SPLINE
SPL {X  -146.770, Y  +318.818, Z    +0.000, E1  +325.496, E3 -247483.059}
SPL {X  -156.430, Y  +348.936, Z    +0.000, E1  +338.153, E3 -247499.791}
SPL {X  -159.088, Y  +365.539, Z    +0.000, E1  +347.196, E3 -247504.201}
SPL {X  -159.820, Y  +375.127, Z    +0.000, E1  +353.170, E3 -247505.625}
SPL {X  -159.990, Y  +382.134, Z    +0.000, E1  +357.935, E3 -247506.144}
SPL {X  -159.990, Y  +385.595, Z    +0.000, E1  +360.838, E3 -247506.258}
SPL {X  -159.990, Y  +390.176, Z    +0.000, E1  +366.367, E3 -247506.527}
SPL {X  -159.990, Y  +395.747, Z    +0.000, E1  +374.484, E3 -247507.153}
SPL {X  -159.990, Y  +402.387, Z    +0.000, E1  +384.140, E3 -247508.385}
SPL {X  -159.990, Y  +414.244, Z    +0.000, E1  +397.704, E3 -247512.018}
SPL {X  -159.990, Y  +460.468, Z    +0.000, E1  +416.751, E3 -247536.110}
SPL {X  -159.990, Y  +537.348, Z    +0.000, E1  +420.157, E3 -247606.121}
SPL {X  -159.990, Y  +545.972, Z    +0.000, E1  +420.143, E3 -247616.656}
SPL {X  -159.990, Y  +557.131, Z    +0.000, E1  +420.184, E3 -247630.170}
SPL {X  -159.990, Y  +569.073, Z    +0.000, E1  +420.153, E3 -247644.764}
SPL {X  -159.990, Y  +577.562, Z    +0.000, E1  +420.146, E3 -247655.104}
SPL {X  -159.990, Y  +585.415, Z    +0.000, E1  +420.147, E3 -247664.670}
SPL {X  -159.990, Y  +594.125, Z    +0.000, E1  +420.153, E3 -247675.256}
SPL {X  -159.990, Y  +602.716, Z    +0.000, E1  +420.150, E3 -247685.719}
SPL {X  -159.990, Y  +612.205, Z    +0.000, E1  +420.159, E3 -247697.255}
SPL {X  -159.990, Y  +624.752, Z    +0.000, E1  +420.194, E3 -247712.463}
SPL {X  -159.990, Y  +640.062, Z    +0.000, E1  +420.188, E3 -247731.127}
SPL {X  -159.990, Y  +652.098, Z    +0.000, E1  +420.153, E3 -247745.837}
SPL {X  -159.990, Y  +661.466, Z    +0.000, E1  +420.154, E3 -247757.248}
SPL {X  -159.963, Y  +674.441, Z    +0.000, E1  +420.189, E3 -247772.999}
SPL {X  -159.339, Y  +685.922, Z    +0.000, E1  +420.057, E3 -247787.677}
SPL {X  -158.381, Y  +694.132, Z    +0.000, E1  +419.909, E3 -247798.675}
SPL {X  -157.192, Y  +701.291, Z    +0.000, E1  +419.715, E3 -247808.645}
SPL {X  -155.426, Y  +709.440, Z    +0.000, E1  +419.459, E3 -247820.343}
SPL {X  -153.239, Y  +717.485, Z    +0.000, E1  +419.087, E3 -247832.388}
SPL {X  -150.608, Y  +725.483, Z    +0.000, E1  +418.677, E3 -247844.733}
SPL {X  -148.008, Y  +732.249, Z    +0.000, E1  +418.192, E3 -247855.600}
SPL {X  -145.943, Y  +737.055, Z    +0.000, E1  +417.829, E3 -247863.458}
SPL {X  -143.898, Y  +741.430, Z    +0.000, E1  +417.467, E3 -247870.728}
SPL {X  -140.579, Y  +747.882, Z    +0.000, E1  +416.895, E3 -247881.607}
SPL {X  -137.120, Y  +753.931, Z    +0.000, E1  +416.213, E3 -247892.067}
SPL {X  -120.054, Y  +777.254, Z    +0.000, E1  +409.463, E3 -247978.813}
ENDSPLINE

SPLINE
SPL {X  -141.034, Y  +747.040, Z    +0.000, E1  +398.619, E3 -248086.975}
SPL {X  -152.334, Y  +720.400, Z    +0.000, E1  +389.143, E3 -248106.429}
SPL {X  -157.190, Y  +701.303, Z    +0.000, E1  +380.164, E3 -248113.590}
SPL {X  -159.117, Y  +688.191, Z    +0.000, E1  +372.748, E3 -248116.622}
SPL {X  -159.875, Y  +677.561, Z    +0.000, E1  +366.083, E3 -248118.011}
SPL {X  -159.990, Y  +671.043, Z    +0.000, E1  +361.371, E3 -248118.415}
SPL {X  -159.990, Y  +669.269, Z    +0.000, E1  +359.855, E3 -248118.460}
SPL {X  -159.990, Y  +666.850, Z    +0.000, E1  +357.321, E3 -248118.543}
SPL {X  -159.990, Y  +662.495, Z    +0.000, E1  +351.318, E3 -248118.837}
SPL {X  -159.990, Y  +657.714, Z    +0.000, E1  +344.114, E3 -248119.398}
SPL {X  -159.990, Y  +651.822, Z    +0.000, E1  +335.261, E3 -248120.367}
SPL {X  -159.990, Y  +641.369, Z    +0.000, E1  +322.665, E3 -248123.205}
SPL {X  -159.990, Y  +598.251, Z    +0.000, E1  +304.104, E3 -248146.976}
SPL {X  -159.990, Y  +514.954, Z    +0.000, E1  +299.688, E3 -248220.772}
SPL {X  -159.990, Y  +505.641, Z    +0.000, E1  +299.707, E3 -248232.081}
SPL {X  -159.990, Y  +498.210, Z    +0.000, E1  +299.707, E3 -248241.074}
SPL {X  -159.990, Y  +488.988, Z    +0.000, E1  +299.693, E3 -248252.211}
SPL {X  -159.990, Y  +478.987, Z    +0.000, E1  +299.694, E3 -248264.314}
SPL {X  -159.990, Y  +468.796, Z    +0.000, E1  +299.698, E3 -248276.657}
SPL {X  -159.990, Y  +460.399, Z    +0.000, E1  +299.707, E3 -248286.834}
SPL {X  -159.990, Y  +453.289, Z    +0.000, E1  +299.707, E3 -248295.440}
SPL {X  -159.990, Y  +443.890, Z    +0.000, E1  +299.691, E3 -248306.793}
SPL {X  -159.990, Y  +437.910, Z    +0.000, E1  +300.175, E3 -248317.264}
ENDSPLINE

SPLINE
SPL {X  -159.990, Y  +447.165, Z    +0.000, E1  +303.287, E3 -248325.819}
ENDSPLINE

SPLINE
SPL {X  -159.990, Y  +436.354, Z    +0.000, E1  +302.683, E3 -248336.831}
SPL {X  -159.990, Y  +425.140, Z    +0.000, E1  +301.982, E3 -248347.266}
SPL {X  -159.990, Y  +412.625, Z    +0.000, E1  +301.150, E3 -248358.102}
SPL {X  -159.990, Y  +398.951, Z    +0.000, E1  +300.353, E3 -248369.973}
SPL {X  -159.990, Y  +389.564, Z    +0.000, E1  +300.093, E3 -248379.787}
SPL {X  -159.985, Y  +381.230, Z    +0.000, E1  +300.090, E3 -248390.054}
SPL {X  -159.702, Y  +372.900, Z    +0.000, E1  +300.135, E3 -248400.591}
SPL {X  -159.030, Y  +365.001, Z    +0.000, E1  +300.230, E3 -248410.994}
SPL {X  -158.029, Y  +357.528, Z    +0.000, E1  +300.403, E3 -248421.250}
SPL {X  -156.953, Y  +351.476, Z    +0.000, E1  +300.570, E3 -248429.803}
SPL {X  -155.503, Y  +344.875, Z    +0.000, E1  +300.798, E3 -248439.412}
SPL {X  -153.622, Y  +337.813, Z    +0.000, E1  +301.097, E3 -248450.006}
SPL {X  -151.786, Y  +331.925, Z    +0.000, E1  +301.419, E3 -248459.127}
SPL {X  -150.141, Y  +327.233, Z    +0.000, E1  +301.695, E3 -248466.535}
SPL {X  -148.134, Y  +322.059, Z    +0.000, E1  +302.038, E3 -248474.869}
SPL {X  -145.832, Y  +316.699, Z    +0.000, E1  +302.442, E3 -248483.703}
SPL {X  -143.160, Y  +311.071, Z    +0.000, E1  +302.918, E3 -248493.149}
SPL {X  -140.427, Y  +305.839, Z    +0.000, E1  +303.430, E3 -248502.110}
SPL {X  -137.611, Y  +300.891, Z    +0.000, E1  +303.950, E3 -248510.686}
SPL {X  -121.335, Y  +278.219, Z    +0.000, E1  +311.699, E3 -248609.032}
ENDSPLINE

SPLINE
SPL {X  -146.770, Y  +318.818, Z    +0.000, E1  +325.496, E3 -248708.866}
SPL {X  -156.430, Y  +348.936, Z    +0.000, E1  +338.153, E3 -248725.597}
SPL {X  -159.088, Y  +365.539, Z    +0.000, E1  +347.196, E3 -248730.008}
SPL {X  -159.921, Y  +377.798, Z    +0.000, E1  +354.872, E3 -248731.668}
SPL {X  -159.990, Y  +383.148, Z    +0.000, E1  +358.786, E3 -248731.996}
SPL {X  -159.990, Y  +384.761, Z    +0.000, E1  +360.138, E3 -248732.040}
SPL {X  -159.990, Y  +387.385, Z    +0.000, E1  +362.811, E3 -248732.142}
SPL {X  -159.990, Y  +391.439, Z    +0.000, E1  +368.259, E3 -248732.438}
SPL {X  -159.990, Y  +395.747, Z    +0.000, E1  +374.484, E3 -248732.959}
SPL {X  -159.990, Y  +402.387, Z    +0.000, E1  +384.140, E3 -248734.192}
SPL {X  -159.990, Y  +414.244, Z    +0.000, E1  +397.704, E3 -248737.825}
SPL {X  -159.990, Y  +460.468, Z    +0.000, E1  +416.751, E3 -248761.916}
SPL {X  -159.990, Y  +537.348, Z    +0.000, E1  +420.157, E3 -248831.928}
SPL {X  -159.990, Y  +549.907, Z    +0.000, E1  +420.183, E3 -248847.186}
SPL {X  -159.990, Y  +560.677, Z    +0.000, E1  +420.145, E3 -248860.357}
SPL {X  -159.990, Y  +569.073, Z    +0.000, E1  +420.153, E3 -248870.571}
SPL {X  -159.990, Y  +577.562, Z    +0.000, E1  +420.146, E3 -248880.911}
SPL {X  -159.990, Y  +585.415, Z    +0.000, E1  +420.147, E3 -248890.476}
SPL {X  -159.990, Y  +594.125, Z    +0.000, E1  +420.153, E3 -248901.063}
SPL {X  -159.990, Y  +602.716, Z    +0.000, E1  +420.150, E3 -248911.525}
SPL {X  -159.990, Y  +612.205, Z    +0.000, E1  +420.159, E3 -248923.062}
SPL {X  -159.990, Y  +620.604, Z    +0.000, E1  +420.153, E3 -248933.277}
SPL {X  -159.990, Y  +632.106, Z    +0.000, E1  +420.183, E3 -248947.254}
SPL {X  -159.990, Y  +643.341, Z    +0.000, E1  +420.148, E3 -248960.998}
SPL {X  -159.990, Y  +652.098, Z    +0.000, E1  +420.153, E3 -248971.643}
SPL {X  -159.990, Y  +661.466, Z    +0.000, E1  +420.154, E3 -248983.054}
SPL {X  -159.990, Y  +670.781, Z    +0.000, E1  +420.150, E3 -248994.402}
SPL {X  -159.839, Y  +678.445, Z    +0.000, E1  +420.123, E3 -249003.881}
SPL {X  -159.339, Y  +685.922, Z    +0.000, E1  +420.057, E3 -249013.484}
SPL {X  -158.381, Y  +694.132, Z    +0.000, E1  +419.909, E3 -249024.481}
SPL {X  -157.192, Y  +701.291, Z    +0.000, E1  +419.715, E3 -249034.451}
SPL {X  -155.426, Y  +709.440, Z    +0.000, E1  +419.459, E3 -249046.149}
SPL {X  -153.239, Y  +717.485, Z    +0.000, E1  +419.087, E3 -249058.194}
SPL {X  -151.467, Y  +723.022, Z    +0.000, E1  +418.780, E3 -249066.747}
SPL {X  -148.791, Y  +730.306, Z    +0.000, E1  +418.370, E3 -249078.212}
SPL {X  -145.943, Y  +737.055, Z    +0.000, E1  +417.829, E3 -249089.265}
SPL {X  -143.898, Y  +741.430, Z    +0.000, E1  +417.467, E3 -249096.534}
SPL {X  -141.624, Y  +745.927, Z    +0.000, E1  +417.045, E3 -249104.129}
SPL {X  -139.581, Y  +749.692, Z    +0.000, E1  +416.662, E3 -249110.576}
SPL {X  -137.120, Y  +753.931, Z    +0.000, E1  +416.213, E3 -249117.873}
SPL {X  -120.054, Y  +777.254, Z    +0.000, E1  +409.463, E3 -249204.619}
ENDSPLINE

SPLINE
SPL {X  -141.034, Y  +747.040, Z    +0.000, E1  +398.619, E3 -249312.781}
SPL {X  -152.334, Y  +720.400, Z    +0.000, E1  +389.143, E3 -249332.236}
SPL {X  -157.190, Y  +701.303, Z    +0.000, E1  +380.164, E3 -249339.396}
SPL {X  -159.117, Y  +688.191, Z    +0.000, E1  +372.748, E3 -249342.428}
SPL {X  -159.875, Y  +677.561, Z    +0.000, E1  +366.083, E3 -249343.818}
SPL {X  -159.990, Y  +669.975, Z    +0.000, E1  +360.595, E3 -249344.249}
SPL {X  -159.990, Y  +666.850, Z    +0.000, E1  +357.321, E3 -249344.349}
SPL {X  -159.990, Y  +662.495, Z    +0.000, E1  +351.318, E3 -249344.644}
SPL {X  -159.990, Y  +657.714, Z    +0.000, E1  +344.114, E3 -249345.205}
SPL {X  -159.990, Y  +651.822, Z    +0.000, E1  +335.261, E3 -249346.173}
SPL {X  -159.990, Y  +641.369, Z    +0.000, E1  +322.665, E3 -249349.011}
SPL {X  -159.990, Y  +598.251, Z    +0.000, E1  +304.104, E3 -249372.782}
SPL {X  -159.990, Y  +514.954, Z    +0.000, E1  +299.688, E3 -249446.578}
SPL {X  -159.990, Y  +505.641, Z    +0.000, E1  +299.707, E3 -249457.887}
SPL {X  -159.990, Y  +498.210, Z    +0.000, E1  +299.707, E3 -249466.881}
SPL {X  -159.990, Y  +488.988, Z    +0.000, E1  +299.693, E3 -249478.017}
SPL {X  -159.990, Y  +478.987, Z    +0.000, E1  +299.694, E3 -249490.120}
SPL {X  -159.990, Y  +468.796, Z    +0.000, E1  +299.698, E3 -249502.464}
SPL {X  -159.990, Y  +460.399, Z    +0.000, E1  +299.707, E3 -249512.641}
SPL {X  -159.990, Y  +453.289, Z    +0.000, E1  +299.707, E3 -249521.246}
SPL {X  -159.990, Y  +443.890, Z    +0.000, E1  +299.691, E3 -249532.600}
SPL {X  -159.990, Y  +437.910, Z    +0.000, E1  +300.175, E3 -249543.070}
ENDSPLINE

SPLINE
SPL {X  -159.990, Y  +447.165, Z    +0.000, E1  +303.287, E3 -249551.626}
ENDSPLINE

SPLINE
SPL {X  -159.990, Y  +436.354, Z    +0.000, E1  +302.683, E3 -249562.637}
SPL {X  -159.990, Y  +425.140, Z    +0.000, E1  +301.982, E3 -249573.072}
SPL {X  -159.990, Y  +412.625, Z    +0.000, E1  +301.150, E3 -249583.908}
SPL {X  -159.990, Y  +398.951, Z    +0.000, E1  +300.353, E3 -249595.780}
SPL {X  -159.990, Y  +389.564, Z    +0.000, E1  +300.093, E3 -249605.594}
SPL {X  -159.985, Y  +381.230, Z    +0.000, E1  +300.090, E3 -249615.861}
SPL {X  -159.702, Y  +372.900, Z    +0.000, E1  +300.135, E3 -249626.398}
SPL {X  -159.030, Y  +365.001, Z    +0.000, E1  +300.230, E3 -249636.801}
SPL {X  -157.449, Y  +354.098, Z    +0.000, E1  +300.447, E3 -249651.800}
SPL {X  -155.503, Y  +344.875, Z    +0.000, E1  +300.798, E3 -249665.219}
SPL {X  -153.622, Y  +337.813, Z    +0.000, E1  +301.097, E3 -249675.812}
SPL {X  -150.877, Y  +329.275, Z    +0.000, E1  +301.527, E3 -249689.037}
SPL {X  -148.134, Y  +322.059, Z    +0.000, E1  +302.038, E3 -249700.675}
SPL {X  -145.832, Y  +316.699, Z    +0.000, E1  +302.442, E3 -249709.510}
SPL {X  -143.160, Y  +311.071, Z    +0.000, E1  +302.918, E3 -249718.955}
SPL {X  -140.427, Y  +305.839, Z    +0.000, E1  +303.430, E3 -249727.916}
SPL {X  -137.611, Y  +300.891, Z    +0.000, E1  +303.950, E3 -249736.492}
SPL {X  -121.335, Y  +278.219, Z    +0.000, E1  +311.699, E3 -249834.838}
ENDSPLINE

SPLINE
SPL {X  -146.770, Y  +318.818, Z    +0.000, E1  +325.496, E3 -249934.672}
SPL {X  -156.430, Y  +348.936, Z    +0.000, E1  +338.153, E3 -249951.404}
SPL {X  -159.088, Y  +365.539, Z    +0.000, E1  +347.196, E3 -249955.814}
SPL {X  -159.820, Y  +375.127, Z    +0.000, E1  +353.170, E3 -249957.238}
SPL {X  -159.990, Y  +382.134, Z    +0.000, E1  +357.935, E3 -249957.757}
SPL {X  -159.990, Y  +385.595, Z    +0.000, E1  +360.838, E3 -249957.871}
SPL {X  -159.990, Y  +390.176, Z    +0.000, E1  +366.367, E3 -249958.140}
SPL {X  -159.990, Y  +395.747, Z    +0.000, E1  +374.484, E3 -249958.766}
SPL {X  -159.990, Y  +404.190, Z    +0.000, E1  +386.444, E3 -249960.448}
SPL {X  -159.990, Y  +418.143, Z    +0.000, E1  +401.167, E3 -249965.041}
SPL {X  -159.990, Y  +460.468, Z    +0.000, E1  +416.751, E3 -249987.723}
SPL {X  -159.990, Y  +537.348, Z    +0.000, E1  +420.157, E3 -250057.734}
SPL {X  -159.990, Y  +549.907, Z    +0.000, E1  +420.183, E3 -250072.992}
SPL {X  -159.990, Y  +560.677, Z    +0.000, E1  +420.145, E3 -250086.163}
SPL {X  -159.990, Y  +569.073, Z    +0.000, E1  +420.153, E3 -250096.377}
SPL {X  -159.990, Y  +581.828, Z    +0.000, E1  +420.191, E3 -250111.837}
SPL {X  -159.990, Y  +594.125, Z    +0.000, E1  +420.153, E3 -250126.869}
SPL {X  -159.990, Y  +602.716, Z    +0.000, E1  +420.150, E3 -250137.332}
SPL {X  -159.990, Y  +612.205, Z    +0.000, E1  +420.159, E3 -250148.868}
SPL {X  -159.990, Y  +620.604, Z    +0.000, E1  +420.153, E3 -250159.084}
SPL {X  -159.990, Y  +632.106, Z    +0.000, E1  +420.183, E3 -250173.061}
SPL {X  -159.990, Y  +643.341, Z    +0.000, E1  +420.148, E3 -250186.804}
SPL {X  -159.990, Y  +652.098, Z    +0.000, E1  +420.153, E3 -250197.449}
SPL {X  -159.990, Y  +661.466, Z    +0.000, E1  +420.154, E3 -250208.861}
SPL {X  -159.990, Y  +670.781, Z    +0.000, E1  +420.150, E3 -250220.209}
SPL {X  -159.839, Y  +678.445, Z    +0.000, E1  +420.123, E3 -250229.688}
SPL {X  -159.339, Y  +685.922, Z    +0.000, E1  +420.057, E3 -250239.290}
SPL {X  -158.381, Y  +694.132, Z    +0.000, E1  +419.909, E3 -250250.287}
SPL {X  -157.192, Y  +701.291, Z    +0.000, E1  +419.715, E3 -250260.258}
SPL {X  -155.426, Y  +709.440, Z    +0.000, E1  +419.459, E3 -250271.956}
SPL {X  -153.239, Y  +717.485, Z    +0.000, E1  +419.087, E3 -250284.001}
SPL {X  -150.608, Y  +725.483, Z    +0.000, E1  +418.677, E3 -250296.346}
SPL {X  -148.008, Y  +732.249, Z    +0.000, E1  +418.192, E3 -250307.213}
SPL {X  -145.943, Y  +737.055, Z    +0.000, E1  +417.829, E3 -250315.071}
SPL {X  -143.898, Y  +741.430, Z    +0.000, E1  +417.467, E3 -250322.341}
SPL {X  -141.624, Y  +745.927, Z    +0.000, E1  +417.045, E3 -250329.936}
SPL {X  -139.581, Y  +749.692, Z    +0.000, E1  +416.662, E3 -250336.383}
SPL {X  -137.120, Y  +753.931, Z    +0.000, E1  +416.213, E3 -250343.680}
SPL {X  -120.054, Y  +777.254, Z    +0.000, E1  +409.463, E3 -250430.426}
ENDSPLINE

SPLINE
SPL {X  -141.034, Y  +747.040, Z    +0.000, E1  +398.619, E3 -250538.588}
SPL {X  -152.334, Y  +720.400, Z    +0.000, E1  +389.143, E3 -250558.042}
SPL {X  -157.190, Y  +701.303, Z    +0.000, E1  +380.164, E3 -250565.203}
SPL {X  -159.460, Y  +684.516, Z    +0.000, E1  +370.556, E3 -250568.798}
SPL {X  -159.938, Y  +675.597, Z    +0.000, E1  +364.669, E3 -250569.805}
SPL {X  -159.990, Y  +671.043, Z    +0.000, E1  +361.371, E3 -250570.028}
SPL {X  -159.990, Y  +669.269, Z    +0.000, E1  +359.855, E3 -250570.073}
SPL {X  -159.990, Y  +666.850, Z    +0.000, E1  +357.321, E3 -250570.156}
SPL {X  -159.990, Y  +662.495, Z    +0.000, E1  +351.318, E3 -250570.450}
SPL {X  -159.990, Y  +657.714, Z    +0.000, E1  +344.114, E3 -250571.011}
SPL {X  -159.990, Y  +651.822, Z    +0.000, E1  +335.261, E3 -250571.979}
SPL {X  -159.990, Y  +641.369, Z    +0.000, E1  +322.665, E3 -250574.818}
SPL {X  -159.990, Y  +598.251, Z    +0.000, E1  +304.104, E3 -250598.589}
SPL {X  -159.990, Y  +514.954, Z    +0.000, E1  +299.688, E3 -250672.384}
SPL {X  -159.990, Y  +505.641, Z    +0.000, E1  +299.707, E3 -250683.694}
SPL {X  -159.990, Y  +498.210, Z    +0.000, E1  +299.707, E3 -250692.687}
SPL {X  -159.990, Y  +488.988, Z    +0.000, E1  +299.693, E3 -250703.824}
SPL {X  -159.990, Y  +478.987, Z    +0.000, E1  +299.694, E3 -250715.926}
SPL {X  -159.990, Y  +468.796, Z    +0.000, E1  +299.698, E3 -250728.270}
SPL {X  -159.990, Y  +456.606, Z    +0.000, E1  +299.670, E3 -250742.976}
SPL {X  -159.990, Y  +443.890, Z    +0.000, E1  +299.691, E3 -250758.406}
SPL {X  -159.990, Y  +437.910, Z    +0.000, E1  +300.175, E3 -250768.877}
ENDSPLINE

SPLINE
SPL {X  -159.990, Y  +447.165, Z    +0.000, E1  +303.287, E3 -250777.432}
ENDSPLINE

SPLINE
SPL {X  -159.990, Y  +436.354, Z    +0.000, E1  +302.683, E3 -250788.443}
SPL {X  -159.990, Y  +425.140, Z    +0.000, E1  +301.982, E3 -250798.879}
SPL {X  -159.990, Y  +412.625, Z    +0.000, E1  +301.150, E3 -250809.715}
SPL {X  -159.990, Y  +398.951, Z    +0.000, E1  +300.353, E3 -250821.586}
SPL {X  -159.990, Y  +389.564, Z    +0.000, E1  +300.093, E3 -250831.400}
SPL {X  -159.985, Y  +381.230, Z    +0.000, E1  +300.090, E3 -250841.667}
SPL {X  -159.702, Y  +372.900, Z    +0.000, E1  +300.135, E3 -250852.204}
SPL {X  -159.030, Y  +365.001, Z    +0.000, E1  +300.230, E3 -250862.607}
SPL {X  -158.029, Y  +357.528, Z    +0.000, E1  +300.403, E3 -250872.862}
SPL {X  -156.953, Y  +351.476, Z    +0.000, E1  +300.570, E3 -250881.416}
SPL {X  -155.503, Y  +344.875, Z    +0.000, E1  +300.798, E3 -250891.025}
SPL {X  -153.622, Y  +337.813, Z    +0.000, E1  +301.097, E3 -250901.619}
SPL {X  -150.877, Y  +329.275, Z    +0.000, E1  +301.527, E3 -250914.843}
SPL {X  -148.134, Y  +322.059, Z    +0.000, E1  +302.038, E3 -250926.482}
SPL {X  -145.832, Y  +316.699, Z    +0.000, E1  +302.442, E3 -250935.316}
SPL {X  -143.160, Y  +311.071, Z    +0.000, E1  +302.918, E3 -250944.762}
SPL {X  -140.427, Y  +305.839, Z    +0.000, E1  +303.430, E3 -250953.723}
SPL {X  -137.611, Y  +300.891, Z    +0.000, E1  +303.950, E3 -250962.299}
SPL {X  -121.335, Y  +278.219, Z    +0.000, E1  +311.699, E3 -251060.645}
ENDSPLINE

SPLINE
SPL {X  -146.770, Y  +318.818, Z    +0.000, E1  +325.496, E3 -251160.479}
SPL {X  -156.430, Y  +348.936, Z    +0.000, E1  +338.153, E3 -251177.210}
SPL {X  -159.088, Y  +365.539, Z    +0.000, E1  +347.196, E3 -251181.621}
SPL {X  -159.921, Y  +377.798, Z    +0.000, E1  +354.872, E3 -251183.281}
SPL {X  -159.990, Y  +384.169, Z    +0.000, E1  +359.534, E3 -251183.637}
SPL {X  -159.990, Y  +386.366, Z    +0.000, E1  +361.774, E3 -251183.701}
SPL {X  -159.990, Y  +390.176, Z    +0.000, E1  +366.367, E3 -251183.947}
SPL {X  -159.990, Y  +395.747, Z    +0.000, E1  +374.484, E3 -251184.572}
SPL {X  -159.990, Y  +402.387, Z    +0.000, E1  +384.140, E3 -251185.805}
SPL {X  -159.990, Y  +414.244, Z    +0.000, E1  +397.704, E3 -251189.438}
SPL {X  -159.990, Y  +460.468, Z    +0.000, E1  +416.751, E3 -251213.529}
SPL {X  -159.990, Y  +537.348, Z    +0.000, E1  +420.157, E3 -251283.541}
SPL {X  -159.990, Y  +545.972, Z    +0.000, E1  +420.143, E3 -251294.075}
SPL {X  -159.990, Y  +557.131, Z    +0.000, E1  +420.184, E3 -251307.589}
SPL {X  -159.990, Y  +569.073, Z    +0.000, E1  +420.153, E3 -251322.184}
SPL {X  -159.990, Y  +581.828, Z    +0.000, E1  +420.191, E3 -251337.643}
SPL {X  -159.990, Y  +594.125, Z    +0.000, E1  +420.153, E3 -251352.676}
SPL {X  -159.990, Y  +602.716, Z    +0.000, E1  +420.150, E3 -251363.138}
SPL {X  -159.990, Y  +612.205, Z    +0.000, E1  +420.159, E3 -251374.675}
SPL {X  -159.990, Y  +624.752, Z    +0.000, E1  +420.194, E3 -251389.883}
SPL {X  -159.990, Y  +640.062, Z    +0.000, E1  +420.188, E3 -251408.546}
SPL {X  -159.990, Y  +652.098, Z    +0.000, E1  +420.153, E3 -251423.256}
SPL {X  -159.990, Y  +661.466, Z    +0.000, E1  +420.154, E3 -251434.667}
SPL {X  -159.963, Y  +674.441, Z    +0.000, E1  +420.189, E3 -251450.418}
SPL {X  -159.339, Y  +685.922, Z    +0.000, E1  +420.057, E3 -251465.097}
SPL {X  -158.381, Y  +694.132, Z    +0.000, E1  +419.909, E3 -251476.094}
SPL {X  -156.712, Y  +703.719, Z    +0.000, E1  +419.674, E3 -251489.459}
SPL {X  -154.922, Y  +711.450, Z    +0.000, E1  +419.348, E3 -251500.775}
SPL {X  -153.239, Y  +717.485, Z    +0.000, E1  +419.087, E3 -251509.807}
SPL {X  -150.608, Y  +725.483, Z    +0.000, E1  +418.677, E3 -251522.153}
SPL {X  -148.008, Y  +732.249, Z    +0.000, E1  +418.192, E3 -251533.019}
SPL {X  -145.943, Y  +737.055, Z    +0.000, E1  +417.829, E3 -251540.878}
SPL {X  -143.898, Y  +741.430, Z    +0.000, E1  +417.467, E3 -251548.147}
SPL {X  -141.624, Y  +745.927, Z    +0.000, E1  +417.045, E3 -251555.742}
SPL {X  -139.581, Y  +749.692, Z    +0.000, E1  +416.662, E3 -251562.189}
SPL {X  -137.120, Y  +753.931, Z    +0.000, E1  +416.213, E3 -251569.486}
SPL {X  -120.054, Y  +777.254, Z    +0.000, E1  +409.463, E3 -251656.232}
ENDSPLINE

SPLINE
SPL {X  -141.034, Y  +747.040, Z    +0.000, E1  +398.619, E3 -251764.394}
SPL {X  -152.334, Y  +720.400, Z    +0.000, E1  +389.143, E3 -251783.848}
SPL {X  -157.190, Y  +701.303, Z    +0.000, E1  +380.164, E3 -251791.009}
SPL {X  -159.117, Y  +688.191, Z    +0.000, E1  +372.748, E3 -251794.041}
SPL {X  -159.875, Y  +677.561, Z    +0.000, E1  +366.083, E3 -251795.431}
SPL {X  -159.990, Y  +669.975, Z    +0.000, E1  +360.595, E3 -251795.862}
SPL {X  -159.990, Y  +666.850, Z    +0.000, E1  +357.321, E3 -251795.962}
SPL {X  -159.990, Y  +662.495, Z    +0.000, E1  +351.318, E3 -251796.257}
SPL {X  -159.990, Y  +657.714, Z    +0.000, E1  +344.114, E3 -251796.818}
SPL {X  -159.990, Y  +651.822, Z    +0.000, E1  +335.261, E3 -251797.786}
SPL {X  -159.990, Y  +641.369, Z    +0.000, E1  +322.665, E3 -251800.624}
SPL {X  -159.990, Y  +598.251, Z    +0.000, E1  +304.104, E3 -251824.395}
SPL {X  -159.990, Y  +514.954, Z    +0.000, E1  +299.688, E3 -251898.191}
SPL {X  -159.990, Y  +505.641, Z    +0.000, E1  +299.707, E3 -251909.500}
SPL {X  -159.990, Y  +498.210, Z    +0.000, E1  +299.707, E3 -251918.494}
SPL {X  -159.990, Y  +488.988, Z    +0.000, E1  +299.693, E3 -251929.630}
SPL {X  -159.990, Y  +478.987, Z    +0.000, E1  +299.694, E3 -251941.733}
SPL {X  -159.990, Y  +468.796, Z    +0.000, E1  +299.698, E3 -251954.077}
SPL {X  -159.990, Y  +456.606, Z    +0.000, E1  +299.670, E3 -251968.782}
SPL {X  -159.990, Y  +443.890, Z    +0.000, E1  +299.691, E3 -251984.212}
SPL {X  -159.990, Y  +437.910, Z    +0.000, E1  +300.175, E3 -251994.683}
ENDSPLINE

SPLINE
SPL {X  -159.990, Y  +447.165, Z    +0.000, E1  +303.287, E3 -252003.238}
ENDSPLINE

SPLINE
SPL {X  -159.990, Y  +436.354, Z    +0.000, E1  +302.683, E3 -252014.250}
SPL {X  -159.990, Y  +425.140, Z    +0.000, E1  +301.982, E3 -252024.685}
SPL {X  -159.990, Y  +412.625, Z    +0.000, E1  +301.150, E3 -252035.521}
SPL {X  -159.990, Y  +398.951, Z    +0.000, E1  +300.353, E3 -252047.393}
SPL {X  -159.990, Y  +389.564, Z    +0.000, E1  +300.093, E3 -252057.207}
SPL {X  -159.985, Y  +381.230, Z    +0.000, E1  +300.090, E3 -252067.474}
SPL {X  -159.702, Y  +372.900, Z    +0.000, E1  +300.135, E3 -252078.011}
SPL {X  -159.030, Y  +365.001, Z    +0.000, E1  +300.230, E3 -252088.413}
SPL {X  -158.029, Y  +357.528, Z    +0.000, E1  +300.403, E3 -252098.669}
SPL {X  -156.953, Y  +351.476, Z    +0.000, E1  +300.570, E3 -252107.222}
SPL {X  -155.503, Y  +344.875, Z    +0.000, E1  +300.798, E3 -252116.832}
SPL {X  -153.622, Y  +337.813, Z    +0.000, E1  +301.097, E3 -252127.425}
SPL {X  -151.786, Y  +331.925, Z    +0.000, E1  +301.419, E3 -252136.546}
SPL {X  -150.141, Y  +327.233, Z    +0.000, E1  +301.695, E3 -252143.955}
SPL {X  -148.134, Y  +322.059, Z    +0.000, E1  +302.038, E3 -252152.288}
SPL {X  -145.832, Y  +316.699, Z    +0.000, E1  +302.442, E3 -252161.123}
SPL {X  -143.160, Y  +311.071, Z    +0.000, E1  +302.918, E3 -252170.568}
SPL {X  -140.427, Y  +305.839, Z    +0.000, E1  +303.430, E3 -252179.529}
SPL {X  -137.611, Y  +300.891, Z    +0.000, E1  +303.950, E3 -252188.105}
SPL {X  -121.335, Y  +278.219, Z    +0.000, E1  +311.699, E3 -252286.451}
ENDSPLINE

SPLINE
SPL {X  -146.770, Y  +318.818, Z    +0.000, E1  +325.496, E3 -252386.285}
SPL {X  -156.430, Y  +348.936, Z    +0.000, E1  +338.153, E3 -252403.016}
SPL {X  -159.088, Y  +365.539, Z    +0.000, E1  +347.196, E3 -252407.427}
SPL {X  -159.921, Y  +377.798, Z    +0.000, E1  +354.872, E3 -252409.087}
SPL {X  -159.990, Y  +384.169, Z    +0.000, E1  +359.534, E3 -252409.443}
SPL {X  -159.990, Y  +386.366, Z    +0.000, E1  +361.774, E3 -252409.507}
SPL {X  -159.990, Y  +390.176, Z    +0.000, E1  +366.367, E3 -252409.753}
SPL {X  -159.990, Y  +395.747, Z    +0.000, E1  +374.484, E3 -252410.379}
SPL {X  -159.990, Y  +402.387, Z    +0.000, E1  +384.140, E3 -252411.611}
SPL {X  -159.990, Y  +414.244, Z    +0.000, E1  +397.704, E3 -252415.244}
SPL {X  -159.990, Y  +460.468, Z    +0.000, E1  +416.751, E3 -252439.336}
SPL {X  -159.990, Y  +537.348, Z    +0.000, E1  +420.157, E3 -252509.347}
SPL {X  -159.990, Y  +545.972, Z    +0.000, E1  +420.143, E3 -252519.881}
SPL {X  -159.990, Y  +557.131, Z    +0.000, E1  +420.184, E3 -252533.396}
SPL {X  -159.990, Y  +569.073, Z    +0.000, E1  +420.153, E3 -252547.990}
SPL {X  -159.990, Y  +577.562, Z    +0.000, E1  +420.146, E3 -252558.330}
SPL {X  -159.990, Y  +585.415, Z    +0.000, E1  +420.147, E3 -252567.896}
SPL {X  -159.990, Y  +594.125, Z    +0.000, E1  +420.153, E3 -252578.482}
SPL {X  -159.990, Y  +602.716, Z    +0.000, E1  +420.150, E3 -252588.945}
SPL {X  -159.990, Y  +612.205, Z    +0.000, E1  +420.159, E3 -252600.481}
SPL {X  -159.990, Y  +624.752, Z    +0.000, E1  +420.194, E3 -252615.689}
SPL {X  -159.990, Y  +640.062, Z    +0.000, E1  +420.188, E3 -252634.353}
SPL {X  -159.990, Y  +652.098, Z    +0.000, E1  +420.153, E3 -252649.062}
SPL {X  -159.990, Y  +661.466, Z    +0.000, E1  +420.154, E3 -252660.474}
SPL {X  -159.990, Y  +670.781, Z    +0.000, E1  +420.150, E3 -252671.821}
SPL {X  -159.839, Y  +678.445, Z    +0.000, E1  +420.123, E3 -252681.301}
SPL {X  -159.339, Y  +685.922, Z    +0.000, E1  +420.057, E3 -252690.903}
SPL {X  -158.381, Y  +694.132, Z    +0.000, E1  +419.909, E3 -252701.900}
SPL {X  -156.712, Y  +703.719, Z    +0.000, E1  +419.674, E3 -252715.265}
SPL {X  -154.922, Y  +711.450, Z    +0.000, E1  +419.348, E3 -252726.581}
SPL {X  -153.239, Y  +717.485, Z    +0.000, E1  +419.087, E3 -252735.614}
SPL {X  -150.608, Y  +725.483, Z    +0.000, E1  +418.677, E3 -252747.959}
SPL {X  -148.008, Y  +732.249, Z    +0.000, E1  +418.192, E3 -252758.826}
SPL {X  -145.943, Y  +737.055, Z    +0.000, E1  +417.829, E3 -252766.684}
SPL {X  -143.898, Y  +741.430, Z    +0.000, E1  +417.467, E3 -252773.954}
SPL {X  -141.624, Y  +745.927, Z    +0.000, E1  +417.045, E3 -252781.549}
SPL {X  -139.581, Y  +749.692, Z    +0.000, E1  +416.662, E3 -252787.995}
SPL {X  -137.120, Y  +753.931, Z    +0.000, E1  +416.213, E3 -252795.293}
SPL {X  -120.054, Y  +777.254, Z    +0.000, E1  +409.463, E3 -252882.039}
ENDSPLINE

SPLINE
SPL {X  -141.034, Y  +747.040, Z    +0.000, E1  +398.619, E3 -252990.201}
SPL {X  -152.334, Y  +720.400, Z    +0.000, E1  +389.143, E3 -253009.655}
SPL {X  -157.190, Y  +701.303, Z    +0.000, E1  +380.164, E3 -253016.816}
SPL {X  -159.117, Y  +688.191, Z    +0.000, E1  +372.748, E3 -253019.848}
SPL {X  -159.875, Y  +677.561, Z    +0.000, E1  +366.083, E3 -253021.237}
SPL {X  -159.990, Y  +671.043, Z    +0.000, E1  +361.371, E3 -253021.641}
SPL {X  -159.990, Y  +668.657, Z    +0.000, E1  +359.332, E3 -253021.702}
SPL {X  -159.990, Y  +665.812, Z    +0.000, E1  +355.875, E3 -253021.813}
SPL {X  -159.990, Y  +662.495, Z    +0.000, E1  +351.318, E3 -253022.063}
SPL {X  -159.990, Y  +657.714, Z    +0.000, E1  +344.114, E3 -253022.624}
SPL {X  -159.990, Y  +651.822, Z    +0.000, E1  +335.261, E3 -253023.592}
SPL {X  -159.990, Y  +641.369, Z    +0.000, E1  +322.665, E3 -253026.431}
SPL {X  -159.990, Y  +598.251, Z    +0.000, E1  +304.104, E3 -253050.202}
SPL {X  -159.990, Y  +514.954, Z    +0.000, E1  +299.688, E3 -253123.997}
SPL {X  -159.990, Y  +505.641, Z    +0.000, E1  +299.707, E3 -253135.306}
SPL {X  -159.990, Y  +498.210, Z    +0.000, E1  +299.707, E3 -253144.300}
SPL {X  -159.990, Y  +488.988, Z    +0.000, E1  +299.693, E3 -253155.437}
SPL {X  -159.990, Y  +478.987, Z    +0.000, E1  +299.694, E3 -253167.539}
SPL {X  -159.990, Y  +468.796, Z    +0.000, E1  +299.698, E3 -253179.883}
SPL {X  -159.990, Y  +456.606, Z    +0.000, E1  +299.670, E3 -253194.589}
SPL {X  -159.990, Y  +443.890, Z    +0.000, E1  +299.691, E3 -253210.019}
SPL {X  -159.990, Y  +437.910, Z    +0.000, E1  +300.175, E3 -253220.490}
ENDSPLINE

SPLINE
SPL {X  -159.990, Y  +447.165, Z    +0.000, E1  +303.287, E3 -253229.045}
ENDSPLINE

SPLINE
SPL {X  -159.990, Y  +436.354, Z    +0.000, E1  +302.683, E3 -253240.056}
SPL {X  -159.990, Y  +425.140, Z    +0.000, E1  +301.982, E3 -253250.492}
SPL {X  -159.990, Y  +412.625, Z    +0.000, E1  +301.150, E3 -253261.328}
SPL {X  -159.990, Y  +398.951, Z    +0.000, E1  +300.353, E3 -253273.199}
SPL {X  -159.990, Y  +389.564, Z    +0.000, E1  +300.093, E3 -253283.013}
SPL {X  -159.985, Y  +381.230, Z    +0.000, E1  +300.090, E3 -253293.280}
SPL {X  -159.702, Y  +372.900, Z    +0.000, E1  +300.135, E3 -253303.817}
SPL {X  -159.030, Y  +365.001, Z    +0.000, E1  +300.230, E3 -253314.220}
SPL {X  -157.449, Y  +354.098, Z    +0.000, E1  +300.447, E3 -253329.220}
SPL {X  -155.503, Y  +344.875, Z    +0.000, E1  +300.798, E3 -253342.638}
SPL {X  -153.622, Y  +337.813, Z    +0.000, E1  +301.097, E3 -253353.231}
SPL {X  -150.877, Y  +329.275, Z    +0.000, E1  +301.527, E3 -253366.456}
SPL {X  -148.134, Y  +322.059, Z    +0.000, E1  +302.038, E3 -253378.095}
SPL {X  -145.832, Y  +316.699, Z    +0.000, E1  +302.442, E3 -253386.929}
SPL {X  -143.160, Y  +311.071, Z    +0.000, E1  +302.918, E3 -253396.374}
SPL {X  -140.427, Y  +305.839, Z    +0.000, E1  +303.430, E3 -253405.336}
SPL {X  -137.611, Y  +300.891, Z    +0.000, E1  +303.950, E3 -253413.912}
SPL {X  -121.335, Y  +278.219, Z    +0.000, E1  +311.699, E3 -253512.258}
ENDSPLINE

SPLINE
SPL {X  -146.770, Y  +318.818, Z    +0.000, E1  +325.496, E3 -253612.092}
SPL {X  -156.430, Y  +348.936, Z    +0.000, E1  +338.153, E3 -253628.823}
SPL {X  -159.088, Y  +365.539, Z    +0.000, E1  +347.196, E3 -253633.234}
SPL {X  -159.820, Y  +375.127, Z    +0.000, E1  +353.170, E3 -253634.657}
SPL {X  -159.990, Y  +382.134, Z    +0.000, E1  +357.935, E3 -253635.176}
SPL {X  -159.990, Y  +385.595, Z    +0.000, E1  +360.838, E3 -253635.291}
SPL {X  -159.990, Y  +390.176, Z    +0.000, E1  +366.367, E3 -253635.560}
SPL {X  -159.990, Y  +395.747, Z    +0.000, E1  +374.484, E3 -253636.185}
SPL {X  -159.990, Y  +402.387, Z    +0.000, E1  +384.140, E3 -253637.418}
SPL {X  -159.990, Y  +413.408, Z    +0.000, E1  +396.965, E3 -253640.719}
SPL {X  -159.990, Y  +455.723, Z    +0.000, E1  +415.803, E3 -253662.561}
SPL {X  -159.990, Y  +537.348, Z    +0.000, E1  +420.157, E3 -253735.154}
SPL {X  -159.990, Y  +545.972, Z    +0.000, E1  +420.143, E3 -253745.688}
SPL {X  -159.990, Y  +557.131, Z    +0.000, E1  +420.184, E3 -253759.202}
SPL {X  -159.990, Y  +569.073, Z    +0.000, E1  +420.153, E3 -253773.797}
SPL {X  -159.990, Y  +577.562, Z    +0.000, E1  +420.146, E3 -253784.137}
SPL {X  -159.990, Y  +585.415, Z    +0.000, E1  +420.147, E3 -253793.702}
SPL {X  -159.990, Y  +594.125, Z    +0.000, E1  +420.153, E3 -253804.289}
SPL {X  -159.990, Y  +602.716, Z    +0.000, E1  +420.150, E3 -253814.751}
SPL {X  -159.990, Y  +612.205, Z    +0.000, E1  +420.159, E3 -253826.288}
SPL {X  -159.990, Y  +620.604, Z    +0.000, E1  +420.153, E3 -253836.503}
SPL {X  -159.990, Y  +632.106, Z    +0.000, E1  +420.183, E3 -253850.480}
SPL {X  -159.990, Y  +643.341, Z    +0.000, E1  +420.148, E3 -253864.224}
SPL {X  -159.990, Y  +652.098, Z    +0.000, E1  +420.153, E3 -253874.869}
SPL {X  -159.990, Y  +661.466, Z    +0.000, E1  +420.154, E3 -253886.280}
SPL {X  -159.963, Y  +674.441, Z    +0.000, E1  +420.189, E3 -253902.031}
SPL {X  -159.339, Y  +685.922, Z    +0.000, E1  +420.057, E3 -253916.710}
SPL {X  -158.381, Y  +694.132, Z    +0.000, E1  +419.909, E3 -253927.707}
SPL {X  -156.712, Y  +703.719, Z    +0.000, E1  +419.674, E3 -253941.072}
SPL {X  -154.922, Y  +711.450, Z    +0.000, E1  +419.348, E3 -253952.388}
SPL {X  -153.239, Y  +717.485, Z    +0.000, E1  +419.087, E3 -253961.420}
SPL {X  -150.608, Y  +725.483, Z    +0.000, E1  +418.677, E3 -253973.766}
SPL {X  -148.008, Y  +732.249, Z    +0.000, E1  +418.192, E3 -253984.632}
SPL {X  -145.943, Y  +737.055, Z    +0.000, E1  +417.829, E3 -253992.491}
SPL {X  -143.898, Y  +741.430, Z    +0.000, E1  +417.467, E3 -253999.760}
SPL {X  -140.579, Y  +747.882, Z    +0.000, E1  +416.895, E3 -254010.639}
SPL {X  -137.120, Y  +753.931, Z    +0.000, E1  +416.213, E3 -254021.099}
SPL {X  -120.054, Y  +777.254, Z    +0.000, E1  +409.463, E3 -254107.845}
ENDSPLINE

SPLINE
SPL {X  -141.034, Y  +747.040, Z    +0.000, E1  +398.619, E3 -254216.007}
SPL {X  -152.334, Y  +720.400, Z    +0.000, E1  +389.143, E3 -254235.461}
SPL {X  -157.190, Y  +701.303, Z    +0.000, E1  +380.164, E3 -254242.622}
SPL {X  -159.117, Y  +688.191, Z    +0.000, E1  +372.748, E3 -254245.654}
SPL {X  -159.875, Y  +677.561, Z    +0.000, E1  +366.083, E3 -254247.044}
SPL {X  -159.990, Y  +671.043, Z    +0.000, E1  +361.371, E3 -254247.448}
SPL {X  -159.990, Y  +668.657, Z    +0.000, E1  +359.332, E3 -254247.508}
SPL {X  -159.990, Y  +665.812, Z    +0.000, E1  +355.875, E3 -254247.620}
SPL {X  -159.990, Y  +662.495, Z    +0.000, E1  +351.318, E3 -254247.869}
SPL {X  -159.990, Y  +657.714, Z    +0.000, E1  +344.114, E3 -254248.431}
SPL {X  -159.990, Y  +651.822, Z    +0.000, E1  +335.261, E3 -254249.399}
SPL {X  -159.990, Y  +641.369, Z    +0.000, E1  +322.665, E3 -254252.237}
SPL {X  -159.990, Y  +598.251, Z    +0.000, E1  +304.104, E3 -254276.008}
SPL {X  -159.990, Y  +514.954, Z    +0.000, E1  +299.688, E3 -254349.804}
SPL {X  -159.990, Y  +501.679, Z    +0.000, E1  +299.667, E3 -254365.841}
SPL {X  -159.990, Y  +488.988, Z    +0.000, E1  +299.693, E3 -254381.243}
SPL {X  -159.990, Y  +478.987, Z    +0.000, E1  +299.694, E3 -254393.346}
SPL {X  -159.990, Y  +468.796, Z    +0.000, E1  +299.698, E3 -254405.690}
SPL {X  -159.990, Y  +460.399, Z    +0.000, E1  +299.707, E3 -254415.866}
SPL {X  -159.990, Y  +453.289, Z    +0.000, E1  +299.707, E3 -254424.472}
SPL {X  -159.990, Y  +443.890, Z    +0.000, E1  +299.691, E3 -254435.825}
SPL {X  -159.990, Y  +437.910, Z    +0.000, E1  +300.175, E3 -254446.296}
ENDSPLINE

SPLINE
SPL {X  -159.990, Y  +447.165, Z    +0.000, E1  +303.287, E3 -254454.851}
ENDSPLINE

SPLINE
SPL {X  -159.990, Y  +436.354, Z    +0.000, E1  +302.683, E3 -254465.863}
SPL {X  -159.990, Y  +425.140, Z    +0.000, E1  +301.982, E3 -254476.298}
SPL {X  -159.990, Y  +412.625, Z    +0.000, E1  +301.150, E3 -254487.134}
SPL {X  -159.990, Y  +398.951, Z    +0.000, E1  +300.353, E3 -254499.006}
SPL {X  -159.990, Y  +389.564, Z    +0.000, E1  +300.093, E3 -254508.819}
SPL {X  -159.985, Y  +381.230, Z    +0.000, E1  +300.090, E3 -254519.086}
SPL {X  -159.702, Y  +372.900, Z    +0.000, E1  +300.135, E3 -254529.623}
SPL {X  -159.030, Y  +365.001, Z    +0.000, E1  +300.230, E3 -254540.026}
SPL {X  -157.449, Y  +354.098, Z    +0.000, E1  +300.447, E3 -254555.026}
SPL {X  -155.503, Y  +344.875, Z    +0.000, E1  +300.798, E3 -254568.445}
SPL {X  -153.622, Y  +337.813, Z    +0.000, E1  +301.097, E3 -254579.038}
SPL {X  -150.877, Y  +329.275, Z    +0.000, E1  +301.527, E3 -254592.263}
SPL {X  -148.134, Y  +322.059, Z    +0.000, E1  +302.038, E3 -254603.901}
SPL {X  -145.832, Y  +316.699, Z    +0.000, E1  +302.442, E3 -254612.736}
SPL {X  -143.160, Y  +311.071, Z    +0.000, E1  +302.918, E3 -254622.181}
SPL {X  -140.427, Y  +305.839, Z    +0.000, E1  +303.430, E3 -254631.142}
SPL {X  -137.611, Y  +300.891, Z    +0.000, E1  +303.950, E3 -254639.718}
SPL {X  -121.335, Y  +278.219, Z    +0.000, E1  +311.699, E3 -254738.064}
ENDSPLINE

SPLINE
SPL {X  -146.770, Y  +318.818, Z    +0.000, E1  +325.496, E3 -254837.898}
SPL {X  -156.430, Y  +348.936, Z    +0.000, E1  +338.153, E3 -254854.629}
SPL {X  -159.088, Y  +365.539, Z    +0.000, E1  +347.196, E3 -254859.040}
SPL {X  -159.820, Y  +375.127, Z    +0.000, E1  +353.170, E3 -254860.464}
SPL {X  -159.990, Y  +382.134, Z    +0.000, E1  +357.935, E3 -254860.982}
SPL {X  -159.990, Y  +385.595, Z    +0.000, E1  +360.838, E3 -254861.097}
SPL {X  -159.990, Y  +390.176, Z    +0.000, E1  +366.367, E3 -254861.366}
SPL {X  -159.990, Y  +395.747, Z    +0.000, E1  +374.484, E3 -254861.992}
SPL {X  -159.990, Y  +404.190, Z    +0.000, E1  +386.444, E3 -254863.674}
SPL {X  -159.990, Y  +418.143, Z    +0.000, E1  +401.167, E3 -254868.267}
SPL {X  -159.990, Y  +460.468, Z    +0.000, E1  +416.751, E3 -254890.949}
SPL {X  -159.990, Y  +537.348, Z    +0.000, E1  +420.157, E3 -254960.960}
SPL {X  -159.990, Y  +549.907, Z    +0.000, E1  +420.183, E3 -254976.218}
SPL {X  -159.990, Y  +560.677, Z    +0.000, E1  +420.145, E3 -254989.389}
SPL {X  -159.990, Y  +569.073, Z    +0.000, E1  +420.153, E3 -254999.603}
SPL {X  -159.990, Y  +581.828, Z    +0.000, E1  +420.191, E3 -255015.062}
SPL {X  -159.990, Y  +594.125, Z    +0.000, E1  +420.153, E3 -255030.095}
SPL {X  -159.990, Y  +602.716, Z    +0.000, E1  +420.150, E3 -255040.558}
SPL {X  -159.990, Y  +612.205, Z    +0.000, E1  +420.159, E3 -255052.094}
SPL {X  -159.990, Y  +624.752, Z    +0.000, E1  +420.194, E3 -255067.302}
SPL {X  -159.990, Y  +640.062, Z    +0.000, E1  +420.188, E3 -255085.966}
SPL {X  -159.990, Y  +652.098, Z    +0.000, E1  +420.153, E3 -255100.675}
SPL {X  -159.990, Y  +661.466, Z    +0.000, E1  +420.154, E3 -255112.087}
SPL {X  -159.963, Y  +674.441, Z    +0.000, E1  +420.189, E3 -255127.837}
SPL {X  -159.339, Y  +685.922, Z    +0.000, E1  +420.057, E3 -255142.516}
SPL {X  -158.381, Y  +694.132, Z    +0.000, E1  +419.909, E3 -255153.513}
SPL {X  -157.192, Y  +701.291, Z    +0.000, E1  +419.715, E3 -255163.484}
SPL {X  -155.426, Y  +709.440, Z    +0.000, E1  +419.459, E3 -255175.182}
SPL {X  -153.239, Y  +717.485, Z    +0.000, E1  +419.087, E3 -255187.227}
SPL {X  -150.608, Y  +725.483, Z    +0.000, E1  +418.677, E3 -255199.572}
SPL {X  -148.008, Y  +732.249, Z    +0.000, E1  +418.192, E3 -255210.439}
SPL {X  -145.943, Y  +737.055, Z    +0.000, E1  +417.829, E3 -255218.297}
SPL {X  -143.898, Y  +741.430, Z    +0.000, E1  +417.467, E3 -255225.566}
SPL {X  -141.624, Y  +745.927, Z    +0.000, E1  +417.045, E3 -255233.162}
SPL {X  -139.581, Y  +749.692, Z    +0.000, E1  +416.662, E3 -255239.608}
SPL {X  -137.120, Y  +753.931, Z    +0.000, E1  +416.213, E3 -255246.906}
SPL {X  -120.054, Y  +777.254, Z    +0.000, E1  +409.463, E3 -255333.652}
ENDSPLINE

SPLINE
SPL {X  -141.034, Y  +747.040, Z    +0.000, E1  +398.619, E3 -255441.814}
SPL {X  -152.334, Y  +720.400, Z    +0.000, E1  +389.143, E3 -255461.268}
SPL {X  -157.190, Y  +701.303, Z    +0.000, E1  +380.164, E3 -255468.428}
SPL {X  -159.117, Y  +688.191, Z    +0.000, E1  +372.748, E3 -255471.460}
SPL {X  -159.875, Y  +677.561, Z    +0.000, E1  +366.083, E3 -255472.850}
SPL {X  -159.990, Y  +671.043, Z    +0.000, E1  +361.371, E3 -255473.254}
SPL {X  -159.990, Y  +669.269, Z    +0.000, E1  +359.855, E3 -255473.299}
SPL {X  -159.990, Y  +666.850, Z    +0.000, E1  +357.321, E3 -255473.381}
SPL {X  -159.990, Y  +662.495, Z    +0.000, E1  +351.318, E3 -255473.676}
SPL {X  -159.990, Y  +657.714, Z    +0.000, E1  +344.114, E3 -255474.237}
SPL {X  -159.990, Y  +651.822, Z    +0.000, E1  +335.261, E3 -255475.205}
SPL {X  -159.990, Y  +641.369, Z    +0.000, E1  +322.665, E3 -255478.043}
SPL {X  -159.990, Y  +598.251, Z    +0.000, E1  +304.104, E3 -255501.815}
SPL {X  -159.990, Y  +514.954, Z    +0.000, E1  +299.688, E3 -255575.610}
SPL {X  -159.990, Y  +501.679, Z    +0.000, E1  +299.667, E3 -255591.647}
SPL {X  -159.990, Y  +488.988, Z    +0.000, E1  +299.693, E3 -255607.050}
SPL {X  -159.990, Y  +478.987, Z    +0.000, E1  +299.694, E3 -255619.152}
SPL {X  -159.990, Y  +468.796, Z    +0.000, E1  +299.698, E3 -255631.496}
SPL {X  -159.990, Y  +460.399, Z    +0.000, E1  +299.707, E3 -255641.673}
SPL {X  -159.990, Y  +453.289, Z    +0.000, E1  +299.707, E3 -255650.278}
SPL {X  -159.990, Y  +443.890, Z    +0.000, E1  +299.691, E3 -255661.632}
SPL {X  -159.990, Y  +437.910, Z    +0.000, E1  +300.175, E3 -255672.103}
ENDSPLINE

SPLINE
SPL {X  -159.990, Y  +447.165, Z    +0.000, E1  +303.287, E3 -255680.658}
ENDSPLINE

SPLINE
SPL {X  -159.990, Y  +436.354, Z    +0.000, E1  +302.683, E3 -255691.669}
SPL {X  -159.990, Y  +425.140, Z    +0.000, E1  +301.982, E3 -255702.105}
SPL {X  -159.990, Y  +412.625, Z    +0.000, E1  +301.150, E3 -255712.941}
SPL {X  -159.990, Y  +398.951, Z    +0.000, E1  +300.353, E3 -255724.812}
ENDSPLINE

SPLINE
SPL {X  -159.990, Y  +412.486, Z    +0.000, E1  +305.075, E3 -255737.392}
ENDSPLINE

SPLINE
SPL {X  -159.990, Y  +405.235, Z    +0.000, E1  +305.098, E3 -255748.245}
SPL {X  -159.990, Y  +400.284, Z    +0.000, E1  +305.103, E3 -255755.640}
SPL {X  -159.990, Y  +391.119, Z    +0.000, E1  +305.052, E3 -255769.228}
SPL {X  -159.988, Y  +381.720, Z    +0.000, E1  +305.103, E3 -255783.335}
SPL {X  -159.786, Y  +374.425, Z    +0.000, E1  +305.121, E3 -255794.384}
SPL {X  -159.184, Y  +366.462, Z    +0.000, E1  +305.220, E3 -255806.884}
SPL {X  -158.166, Y  +358.413, Z    +0.000, E1  +305.386, E3 -255819.940}
SPL {X  -156.775, Y  +350.586, Z    +0.000, E1  +305.627, E3 -255833.064}
SPL {X  -155.027, Y  +342.959, Z    +0.000, E1  +305.926, E3 -255846.237}
SPL {X  -152.882, Y  +335.340, Z    +0.000, E1  +306.305, E3 -255859.780}
SPL {X  -150.681, Y  +328.723, Z    +0.000, E1  +306.710, E3 -255871.874}
SPL {X  -147.884, Y  +321.449, Z    +0.000, E1  +307.200, E3 -255885.447}
SPL {X  -145.161, Y  +315.232, Z    +0.000, E1  +307.745, E3 -255897.379}
SPL {X  -142.534, Y  +309.830, Z    +0.000, E1  +308.237, E3 -255907.884}
SPL {X  -132.342, Y  +292.599, Z    +0.000, E1  +315.826, E3 -256005.172}
ENDSPLINE

SPLINE
SPL {X  -151.238, Y  +330.309, Z    +0.000, E1  +330.693, E3 -256078.329}
SPL {X  -156.949, Y  +351.453, Z    +0.000, E1  +340.161, E3 -256090.490}
SPL {X  -159.024, Y  +364.945, Z    +0.000, E1  +347.297, E3 -256094.907}
SPL {X  -159.878, Y  +376.512, Z    +0.000, E1  +354.071, E3 -256097.159}
SPL {X  -159.990, Y  +383.659, Z    +0.000, E1  +358.950, E3 -256097.853}
SPL {X  -159.990, Y  +387.327, Z    +0.000, E1  +362.137, E3 -256098.086}
SPL {X  -159.990, Y  +390.622, Z    +0.000, E1  +365.876, E3 -256098.380}
SPL {X  -159.990, Y  +394.493, Z    +0.000, E1  +370.512, E3 -256098.903}
SPL {X  -159.990, Y  +401.377, Z    +0.000, E1  +379.398, E3 -256100.357}
SPL {X  -159.990, Y  +411.365, Z    +0.000, E1  +390.630, E3 -256103.566}
SPL {X  -159.990, Y  +450.467, Z    +0.000, E1  +410.183, E3 -256127.214}
SPL {X  -159.990, Y  +509.934, Z    +0.000, E1  +414.923, E3 -256189.833}
SPL {X  -159.990, Y  +516.848, Z    +0.000, E1  +414.930, E3 -256200.121}
SPL {X  -159.990, Y  +524.818, Z    +0.000, E1  +414.933, E3 -256211.993}
SPL {X  -159.990, Y  +532.100, Z    +0.000, E1  +414.924, E3 -256222.846}
SPL {X  -159.990, Y  +539.391, Z    +0.000, E1  +414.933, E3 -256233.698}
SPL {X  -159.990, Y  +546.283, Z    +0.000, E1  +414.924, E3 -256243.970}
SPL {X  -159.990, Y  +553.734, Z    +0.000, E1  +414.938, E3 -256255.057}
SPL {X  -159.990, Y  +564.956, Z    +0.000, E1  +414.973, E3 -256271.728}
SPL {X  -159.990, Y  +577.902, Z    +0.000, E1  +414.969, E3 -256291.018}
SPL {X  -159.990, Y  +588.063, Z    +0.000, E1  +414.931, E3 -256306.209}
SPL {X  -159.990, Y  +595.273, Z    +0.000, E1  +414.928, E3 -256316.932}
SPL {X  -159.990, Y  +602.326, Z    +0.000, E1  +414.932, E3 -256327.432}
SPL {X  -159.990, Y  +609.708, Z    +0.000, E1  +414.930, E3 -256338.439}
SPL {X  -159.990, Y  +618.088, Z    +0.000, E1  +414.948, E3 -256350.868}
SPL {X  -159.990, Y  +625.928, Z    +0.000, E1  +414.931, E3 -256362.564}
SPL {X  -159.990, Y  +635.803, Z    +0.000, E1  +414.980, E3 -256377.192}
SPL {X  -159.990, Y  +646.303, Z    +0.000, E1  +414.946, E3 -256392.863}
SPL {X  -159.990, Y  +656.335, Z    +0.000, E1  +414.969, E3 -256407.765}
SPL {X  -159.990, Y  +664.577, Z    +0.000, E1  +414.924, E3 -256420.142}
SPL {X  -159.989, Y  +672.128, Z    +0.000, E1  +414.946, E3 -256431.359}
SPL {X  -159.792, Y  +679.466, Z    +0.000, E1  +414.893, E3 -256442.517}
SPL {X  -159.330, Y  +686.016, Z    +0.000, E1  +414.837, E3 -256452.748}
SPL {X  -158.190, Y  +695.432, Z    +0.000, E1  +414.658, E3 -256467.944}
SPL {X  -157.027, Y  +702.151, Z    +0.000, E1  +414.415, E3 -256479.226}
SPL {X  -156.112, Y  +706.513, Z    +0.000, E1  +414.265, E3 -256486.660}
SPL {X  -154.917, Y  +711.470, Z    +0.000, E1  +414.052, E3 -256495.288}
SPL {X  -153.561, Y  +716.398, Z    +0.000, E1  +413.816, E3 -256504.009}
SPL {X  -151.715, Y  +722.287, Z    +0.000, E1  +413.503, E3 -256514.625}
SPL {X  -149.700, Y  +727.952, Z    +0.000, E1  +413.118, E3 -256525.100}
SPL {X  -147.376, Y  +733.767, Z    +0.000, E1  +412.706, E3 -256536.050}
SPL {X  -144.332, Y  +740.529, Z    +0.000, E1  +412.133, E3 -256549.040}
SPL {X  -142.065, Y  +745.081, Z    +0.000, E1  +411.654, E3 -256557.993}
SPL {X  -132.301, Y  +761.463, Z    +0.000, E1  +405.510, E3 -256634.500}
ENDSPLINE

SPLINE
SPL {X  -145.877, Y  +737.201, Z    +0.000, E1  +394.468, E3 -256717.611}
SPL {X  -152.550, Y  +719.721, Z    +0.000, E1  +387.728, E3 -256733.100}
SPL {X  -157.145, Y  +701.536, Z    +0.000, E1  +379.368, E3 -256742.554}
SPL {X  -159.035, Y  +688.952, Z    +0.000, E1  +372.676, E3 -256746.596}
SPL {X  -159.756, Y  +680.154, Z    +0.000, E1  +367.520, E3 -256748.322}
SPL {X  -159.986, Y  +672.560, Z    +0.000, E1  +362.636, E3 -256749.220}
SPL {X  -159.990, Y  +668.344, Z    +0.000, E1  +359.382, E3 -256749.486}
SPL {X  -159.990, Y  +664.070, Z    +0.000, E1  +354.975, E3 -256749.815}
SPL {X  -159.990, Y  +656.953, Z    +0.000, E1  +346.040, E3 -256750.881}
SPL {X  -159.990, Y  +644.589, Z    +0.000, E1  +330.989, E3 -256754.293}
SPL {X  -159.990, Y  +605.095, Z    +0.000, E1  +310.486, E3 -256779.383}
SPL {X  -159.990, Y  +546.155, Z    +0.000, E1  +305.539, E3 -256842.142}
SPL {X  -159.990, Y  +539.348, Z    +0.000, E1  +305.531, E3 -256852.446}
SPL {X  -159.990, Y  +530.752, Z    +0.000, E1  +305.518, E3 -256865.453}
SPL {X  -159.990, Y  +522.797, Z    +0.000, E1  +305.537, E3 -256877.536}
SPL {X  -159.990, Y  +515.332, Z    +0.000, E1  +305.526, E3 -256888.825}
SPL {X  -159.990, Y  +508.047, Z    +0.000, E1  +305.531, E3 -256899.842}
SPL {X  -159.990, Y  +499.403, Z    +0.000, E1  +305.488, E3 -256912.881}
SPL {X  -159.990, Y  +479.413, Z    +0.000, E1  +302.719, E3 -256924.026}
SPL {X  -159.990, Y  +454.926, Z    +0.000, E1  +299.433, E3 -256933.133}
SPL {X  -159.990, Y  +449.697, Z    +0.000, E1  +300.191, E3 -256944.595}
SPL {X  -159.990, Y  +445.847, Z    +0.000, E1  +300.905, E3 -256954.218}
SPL {X  -159.990, Y  +439.266, Z    +0.000, E1  +301.568, E3 -256967.302}
SPL {X  -159.990, Y  +432.883, Z    +0.000, E1  +302.386, E3 -256980.992}
SPL {X  -159.990, Y  +429.044, Z    +0.000, E1  +303.109, E3 -256990.882}
SPL {X  -159.990, Y  +425.222, Z    +0.000, E1  +304.101, E3 -257002.779}
SPL {X  -159.990, Y  +420.083, Z    +0.000, E1  +304.918, E3 -257015.355}
SPL {X  -159.990, Y  +412.567, Z    +0.000, E1  +305.072, E3 -257027.579}
SPL {X  -159.990, Y  +402.790, Z    +0.000, E1  +305.070, E3 -257042.173}
SPL {X  -159.990, Y  +391.119, Z    +0.000, E1  +305.052, E3 -257059.551}
SPL {X  -159.988, Y  +381.720, Z    +0.000, E1  +305.103, E3 -257073.658}
SPL {X  -159.786, Y  +374.425, Z    +0.000, E1  +305.121, E3 -257084.706}
SPL {X  -159.015, Y  +364.863, Z    +0.000, E1  +305.220, E3 -257099.722}
SPL {X  -157.966, Y  +357.131, Z    +0.000, E1  +305.441, E3 -257112.413}
SPL {X  -156.775, Y  +350.586, Z    +0.000, E1  +305.627, E3 -257123.387}
SPL {X  -155.027, Y  +342.959, Z    +0.000, E1  +305.926, E3 -257136.560}
SPL {X  -152.882, Y  +335.340, Z    +0.000, E1  +306.305, E3 -257150.102}
SPL {X  -150.681, Y  +328.723, Z    +0.000, E1  +306.710, E3 -257162.197}
SPL {X  -148.661, Y  +323.366, Z    +0.000, E1  +307.100, E3 -257172.206}
SPL {X  -147.089, Y  +319.560, Z    +0.000, E1  +307.396, E3 -257179.421}
SPL {X  -145.161, Y  +315.232, Z    +0.000, E1  +307.745, E3 -257187.701}
SPL {X  -142.534, Y  +309.830, Z    +0.000, E1  +308.237, E3 -257198.206}
SPL {X  -132.342, Y  +292.599, Z    +0.000, E1  +315.826, E3 -257295.495}
ENDSPLINE

SPLINE
SPL {X  -151.238, Y  +330.309, Z    +0.000, E1  +330.693, E3 -257368.651}
SPL {X  -156.949, Y  +351.453, Z    +0.000, E1  +340.161, E3 -257380.812}
SPL {X  -159.024, Y  +364.945, Z    +0.000, E1  +347.297, E3 -257385.230}
SPL {X  -159.878, Y  +376.512, Z    +0.000, E1  +354.071, E3 -257387.481}
SPL {X  -159.990, Y  +383.659, Z    +0.000, E1  +358.950, E3 -257388.176}
SPL {X  -159.990, Y  +387.327, Z    +0.000, E1  +362.137, E3 -257388.409}
SPL {X  -159.990, Y  +390.622, Z    +0.000, E1  +365.876, E3 -257388.702}
SPL {X  -159.990, Y  +394.493, Z    +0.000, E1  +370.512, E3 -257389.225}
SPL {X  -159.990, Y  +401.377, Z    +0.000, E1  +379.398, E3 -257390.680}
SPL {X  -159.990, Y  +411.365, Z    +0.000, E1  +390.630, E3 -257393.888}
SPL {X  -159.990, Y  +450.467, Z    +0.000, E1  +410.183, E3 -257417.537}
SPL {X  -159.990, Y  +509.934, Z    +0.000, E1  +414.923, E3 -257480.156}
SPL {X  -159.990, Y  +516.848, Z    +0.000, E1  +414.930, E3 -257490.444}
SPL {X  -159.990, Y  +524.818, Z    +0.000, E1  +414.933, E3 -257502.316}
SPL {X  -159.990, Y  +532.100, Z    +0.000, E1  +414.924, E3 -257513.169}
SPL {X  -159.990, Y  +539.391, Z    +0.000, E1  +414.933, E3 -257524.021}
SPL {X  -159.990, Y  +546.283, Z    +0.000, E1  +414.924, E3 -257534.292}
SPL {X  -159.990, Y  +553.734, Z    +0.000, E1  +414.938, E3 -257545.379}
SPL {X  -159.990, Y  +564.956, Z    +0.000, E1  +414.973, E3 -257562.050}
SPL {X  -159.990, Y  +577.902, Z    +0.000, E1  +414.969, E3 -257581.340}
SPL {X  -159.990, Y  +588.063, Z    +0.000, E1  +414.931, E3 -257596.531}
SPL {X  -159.990, Y  +595.273, Z    +0.000, E1  +414.928, E3 -257607.255}
SPL {X  -159.990, Y  +602.326, Z    +0.000, E1  +414.932, E3 -257617.755}
SPL {X  -159.990, Y  +609.708, Z    +0.000, E1  +414.930, E3 -257628.762}
SPL {X  -159.990, Y  +618.088, Z    +0.000, E1  +414.948, E3 -257641.191}
SPL {X  -159.990, Y  +625.928, Z    +0.000, E1  +414.931, E3 -257652.887}
SPL {X  -159.990, Y  +635.803, Z    +0.000, E1  +414.980, E3 -257667.515}
SPL {X  -159.990, Y  +646.303, Z    +0.000, E1  +414.946, E3 -257683.185}
SPL {X  -159.990, Y  +653.312, Z    +0.000, E1  +414.932, E3 -257693.637}
SPL {X  -159.990, Y  +658.943, Z    +0.000, E1  +414.931, E3 -257702.035}
SPL {X  -159.990, Y  +667.151, Z    +0.000, E1  +414.954, E3 -257714.254}
SPL {X  -159.885, Y  +677.285, Z    +0.000, E1  +414.936, E3 -257729.449}
SPL {X  -159.482, Y  +684.244, Z    +0.000, E1  +414.840, E3 -257740.301}
SPL {X  -158.805, Y  +690.934, Z    +0.000, E1  +414.742, E3 -257750.950}
SPL {X  -157.890, Y  +697.337, Z    +0.000, E1  +414.571, E3 -257761.472}
SPL {X  -156.492, Y  +704.774, Z    +0.000, E1  +414.365, E3 -257773.950}
SPL {X  -154.917, Y  +711.470, Z    +0.000, E1  +414.052, E3 -257785.610}
SPL {X  -153.561, Y  +716.398, Z    +0.000, E1  +413.816, E3 -257794.332}
SPL {X  -151.715, Y  +722.287, Z    +0.000, E1  +413.503, E3 -257804.948}
SPL {X  -148.967, Y  +729.859, Z    +0.000, E1  +413.026, E3 -257818.940}
SPL {X  -145.862, Y  +737.236, Z    +0.000, E1  +412.427, E3 -257832.994}
SPL {X  -142.777, Y  +743.691, Z    +0.000, E1  +411.831, E3 -257845.537}
SPL {X  -132.301, Y  +761.463, Z    +0.000, E1  +405.510, E3 -257924.822}
ENDSPLINE

SPLINE
SPL {X  -145.877, Y  +737.201, Z    +0.000, E1  +394.468, E3 -258007.933}
SPL {X  -152.550, Y  +719.721, Z    +0.000, E1  +387.728, E3 -258023.422}
SPL {X  -157.145, Y  +701.536, Z    +0.000, E1  +379.368, E3 -258032.877}
SPL {X  -159.035, Y  +688.952, Z    +0.000, E1  +372.676, E3 -258036.918}
SPL {X  -159.756, Y  +680.154, Z    +0.000, E1  +367.520, E3 -258038.644}
SPL {X  -159.986, Y  +672.560, Z    +0.000, E1  +362.636, E3 -258039.543}
SPL {X  -159.990, Y  +668.344, Z    +0.000, E1  +359.382, E3 -258039.809}
SPL {X  -159.990, Y  +664.070, Z    +0.000, E1  +354.975, E3 -258040.137}
SPL {X  -159.990, Y  +656.953, Z    +0.000, E1  +346.040, E3 -258041.204}
SPL {X  -159.990, Y  +644.589, Z    +0.000, E1  +330.989, E3 -258044.615}
SPL {X  -159.990, Y  +605.095, Z    +0.000, E1  +310.486, E3 -258069.706}
SPL {X  -159.990, Y  +546.155, Z    +0.000, E1  +305.539, E3 -258132.465}
SPL {X  -159.990, Y  +539.348, Z    +0.000, E1  +305.531, E3 -258142.768}
SPL {X  -159.990, Y  +530.752, Z    +0.000, E1  +305.518, E3 -258155.776}
SPL {X  -159.990, Y  +522.797, Z    +0.000, E1  +305.537, E3 -258167.859}
SPL {X  -159.990, Y  +515.332, Z    +0.000, E1  +305.526, E3 -258179.148}
SPL {X  -159.990, Y  +508.047, Z    +0.000, E1  +305.531, E3 -258190.164}
SPL {X  -159.990, Y  +501.296, Z    +0.000, E1  +305.518, E3 -258200.386}
SPL {X  -159.990, Y  +487.558, Z    +0.000, E1  +304.151, E3 -258212.016}
SPL {X  -159.990, Y  +454.926, Z    +0.000, E1  +299.433, E3 -258223.456}
SPL {X  -159.990, Y  +449.697, Z    +0.000, E1  +300.191, E3 -258234.918}
SPL {X  -159.990, Y  +445.847, Z    +0.000, E1  +300.905, E3 -258244.541}
SPL {X  -159.990, Y  +439.266, Z    +0.000, E1  +301.568, E3 -258257.624}
SPL {X  -159.990, Y  +432.883, Z    +0.000, E1  +302.386, E3 -258271.315}
SPL {X  -159.990, Y  +429.044, Z    +0.000, E1  +303.109, E3 -258281.205}
SPL {X  -159.990, Y  +425.222, Z    +0.000, E1  +304.101, E3 -258293.102}
SPL {X  -159.990, Y  +418.562, Z    +0.000, E1  +304.950, E3 -258308.260}
SPL {X  -159.990, Y  +407.911, Z    +0.000, E1  +305.062, E3 -258324.851}
SPL {X  -159.990, Y  +400.284, Z    +0.000, E1  +305.103, E3 -258336.285}
SPL {X  -159.990, Y  +391.119, Z    +0.000, E1  +305.052, E3 -258349.873}
SPL {X  -159.988, Y  +381.720, Z    +0.000, E1  +305.103, E3 -258363.981}
SPL {X  -159.786, Y  +374.425, Z    +0.000, E1  +305.121, E3 -258375.029}
SPL {X  -159.015, Y  +364.863, Z    +0.000, E1  +305.220, E3 -258390.045}
SPL {X  -157.966, Y  +357.131, Z    +0.000, E1  +305.441, E3 -258402.735}
SPL {X  -156.775, Y  +350.586, Z    +0.000, E1  +305.627, E3 -258413.709}
SPL {X  -155.027, Y  +342.959, Z    +0.000, E1  +305.926, E3 -258426.882}
SPL {X  -152.882, Y  +335.340, Z    +0.000, E1  +306.305, E3 -258440.425}
SPL {X  -150.681, Y  +328.723, Z    +0.000, E1  +306.710, E3 -258452.519}
SPL {X  -148.661, Y  +323.366, Z    +0.000, E1  +307.100, E3 -258462.528}
SPL {X  -147.089, Y  +319.560, Z    +0.000, E1  +307.396, E3 -258469.744}
SPL {X  -145.161, Y  +315.232, Z    +0.000, E1  +307.745, E3 -258478.024}
SPL {X  -142.534, Y  +309.830, Z    +0.000, E1  +308.237, E3 -258488.529}
SPL {X  -132.342, Y  +292.599, Z    +0.000, E1  +315.826, E3 -258585.817}
ENDSPLINE

SPLINE
SPL {X  -151.238, Y  +330.309, Z    +0.000, E1  +330.693, E3 -258658.974}
SPL {X  -156.949, Y  +351.453, Z    +0.000, E1  +340.161, E3 -258671.135}
SPL {X  -159.024, Y  +364.945, Z    +0.000, E1  +347.297, E3 -258675.553}
SPL {X  -159.758, Y  +373.891, Z    +0.000, E1  +352.513, E3 -258677.441}
SPL {X  -159.985, Y  +381.208, Z    +0.000, E1  +357.184, E3 -258678.324}
SPL {X  -159.990, Y  +384.493, Z    +0.000, E1  +359.676, E3 -258678.549}
SPL {X  -159.990, Y  +387.327, Z    +0.000, E1  +362.137, E3 -258678.731}
SPL {X  -159.990, Y  +392.053, Z    +0.000, E1  +367.477, E3 -258679.196}
SPL {X  -159.990, Y  +396.158, Z    +0.000, E1  +372.775, E3 -258679.822}
SPL {X  -159.990, Y  +401.377, Z    +0.000, E1  +379.398, E3 -258681.002}
SPL {X  -159.990, Y  +411.365, Z    +0.000, E1  +390.630, E3 -258684.211}
SPL {X  -159.990, Y  +450.467, Z    +0.000, E1  +410.183, E3 -258707.860}
SPL {X  -159.990, Y  +509.934, Z    +0.000, E1  +414.923, E3 -258770.478}
SPL {X  -159.990, Y  +516.848, Z    +0.000, E1  +414.930, E3 -258780.767}
SPL {X  -159.990, Y  +524.818, Z    +0.000, E1  +414.933, E3 -258792.638}
SPL {X  -159.990, Y  +532.100, Z    +0.000, E1  +414.924, E3 -258803.491}
SPL {X  -159.990, Y  +539.391, Z    +0.000, E1  +414.933, E3 -258814.343}
SPL {X  -159.990, Y  +546.283, Z    +0.000, E1  +414.924, E3 -258824.615}
SPL {X  -159.990, Y  +553.734, Z    +0.000, E1  +414.938, E3 -258835.702}
SPL {X  -159.990, Y  +564.956, Z    +0.000, E1  +414.973, E3 -258852.373}
SPL {X  -159.990, Y  +577.902, Z    +0.000, E1  +414.969, E3 -258871.663}
SPL {X  -159.990, Y  +588.063, Z    +0.000, E1  +414.931, E3 -258886.854}
SPL {X  -159.990, Y  +595.273, Z    +0.000, E1  +414.928, E3 -258897.577}
SPL {X  -159.990, Y  +602.326, Z    +0.000, E1  +414.932, E3 -258908.078}
SPL {X  -159.990, Y  +609.708, Z    +0.000, E1  +414.930, E3 -258919.084}
SPL {X  -159.990, Y  +618.088, Z    +0.000, E1  +414.948, E3 -258931.513}
SPL {X  -159.990, Y  +625.928, Z    +0.000, E1  +414.931, E3 -258943.209}
SPL {X  -159.990, Y  +632.991, Z    +0.000, E1  +414.938, E3 -258953.712}
SPL {X  -159.990, Y  +639.033, Z    +0.000, E1  +414.931, E3 -258962.720}
SPL {X  -159.990, Y  +646.303, Z    +0.000, E1  +414.946, E3 -258973.508}
SPL {X  -159.990, Y  +656.335, Z    +0.000, E1  +414.969, E3 -258988.410}
SPL {X  -159.990, Y  +664.577, Z    +0.000, E1  +414.924, E3 -259000.787}
SPL {X  -159.989, Y  +672.128, Z    +0.000, E1  +414.946, E3 -259012.004}
SPL {X  -159.636, Y  +682.136, Z    +0.000, E1  +414.901, E3 -259027.262}
SPL {X  -158.805, Y  +690.934, Z    +0.000, E1  +414.742, E3 -259041.273}
SPL {X  -157.890, Y  +697.337, Z    +0.000, E1  +414.571, E3 -259051.794}
SPL {X  -156.492, Y  +704.774, Z    +0.000, E1  +414.365, E3 -259064.273}
SPL {X  -154.917, Y  +711.470, Z    +0.000, E1  +414.052, E3 -259075.933}
SPL {X  -153.204, Y  +717.603, Z    +0.000, E1  +413.775, E3 -259086.779}
SPL {X  -151.355, Y  +723.351, Z    +0.000, E1  +413.415, E3 -259097.250}
SPL {X  -148.967, Y  +729.859, Z    +0.000, E1  +413.026, E3 -259109.262}
SPL {X  -145.862, Y  +737.236, Z    +0.000, E1  +412.427, E3 -259123.317}
SPL {X  -142.777, Y  +743.691, Z    +0.000, E1  +411.831, E3 -259135.860}
SPL {X  -132.301, Y  +761.463, Z    +0.000, E1  +405.510, E3 -259215.145}
ENDSPLINE

SPLINE
SPL {X  -145.877, Y  +737.201, Z    +0.000, E1  +394.468, E3 -259298.256}
SPL {X  -152.550, Y  +719.721, Z    +0.000, E1  +387.728, E3 -259313.745}
SPL {X  -157.145, Y  +701.536, Z    +0.000, E1  +379.368, E3 -259323.200}
SPL {X  -159.035, Y  +688.952, Z    +0.000, E1  +372.676, E3 -259327.241}
SPL {X  -159.756, Y  +680.154, Z    +0.000, E1  +367.520, E3 -259328.967}
SPL {X  -159.986, Y  +672.560, Z    +0.000, E1  +362.636, E3 -259329.865}
SPL {X  -159.990, Y  +668.344, Z    +0.000, E1  +359.382, E3 -259330.131}
SPL {X  -159.990, Y  +664.070, Z    +0.000, E1  +354.975, E3 -259330.460}
SPL {X  -159.990, Y  +656.953, Z    +0.000, E1  +346.040, E3 -259331.526}
SPL {X  -159.990, Y  +644.589, Z    +0.000, E1  +330.989, E3 -259334.938}
SPL {X  -159.990, Y  +605.095, Z    +0.000, E1  +310.486, E3 -259360.029}
SPL {X  -159.990, Y  +546.155, Z    +0.000, E1  +305.539, E3 -259422.787}
SPL {X  -159.990, Y  +539.348, Z    +0.000, E1  +305.531, E3 -259433.091}
SPL {X  -159.990, Y  +530.752, Z    +0.000, E1  +305.518, E3 -259446.098}
SPL {X  -159.990, Y  +522.797, Z    +0.000, E1  +305.537, E3 -259458.181}
SPL {X  -159.990, Y  +515.332, Z    +0.000, E1  +305.526, E3 -259469.470}
SPL {X  -159.990, Y  +508.047, Z    +0.000, E1  +305.531, E3 -259480.487}
SPL {X  -159.990, Y  +501.296, Z    +0.000, E1  +305.518, E3 -259490.708}
SPL {X  -159.990, Y  +487.558, Z    +0.000, E1  +304.151, E3 -259502.339}
SPL {X  -159.990, Y  +454.926, Z    +0.000, E1  +299.433, E3 -259513.778}
SPL {X  -159.990, Y  +449.697, Z    +0.000, E1  +300.191, E3 -259525.241}
SPL {X  -159.990, Y  +445.847, Z    +0.000, E1  +300.905, E3 -259534.864}
SPL {X  -159.990, Y  +439.266, Z    +0.000, E1  +301.568, E3 -259547.947}
SPL {X  -159.990, Y  +432.883, Z    +0.000, E1  +302.386, E3 -259561.637}
SPL {X  -159.990, Y  +428.299, Z    +0.000, E1  +303.316, E3 -259574.041}
SPL {X  -159.990, Y  +424.402, Z    +0.000, E1  +304.297, E3 -259585.716}
SPL {X  -159.990, Y  +420.083, Z    +0.000, E1  +304.918, E3 -259596.000}
SPL {X  -159.990, Y  +412.567, Z    +0.000, E1  +305.072, E3 -259608.224}
SPL {X  -159.990, Y  +405.235, Z    +0.000, E1  +305.098, E3 -259619.212}
SPL {X  -159.990, Y  +400.284, Z    +0.000, E1  +305.103, E3 -259626.607}
SPL {X  -159.990, Y  +391.119, Z    +0.000, E1  +305.052, E3 -259640.196}
SPL {X  -159.988, Y  +381.720, Z    +0.000, E1  +305.103, E3 -259654.303}
SPL {X  -159.786, Y  +374.425, Z    +0.000, E1  +305.121, E3 -259665.351}
SPL {X  -159.015, Y  +364.863, Z    +0.000, E1  +305.220, E3 -259680.368}
SPL {X  -157.966, Y  +357.131, Z    +0.000, E1  +305.441, E3 -259693.058}
SPL {X  -156.775, Y  +350.586, Z    +0.000, E1  +305.627, E3 -259704.032}
SPL {X  -155.397, Y  +344.442, Z    +0.000, E1  +305.886, E3 -259714.648}
SPL {X  -153.976, Y  +339.046, Z    +0.000, E1  +306.128, E3 -259724.140}
SPL {X  -152.417, Y  +333.859, Z    +0.000, E1  +306.416, E3 -259733.466}
SPL {X  -150.681, Y  +328.723, Z    +0.000, E1  +306.710, E3 -259742.842}
SPL {X  -147.884, Y  +321.449, Z    +0.000, E1  +307.200, E3 -259756.415}
SPL {X  -144.518, Y  +313.862, Z    +0.000, E1  +307.832, E3 -259770.961}
SPL {X  -141.812, Y  +308.430, Z    +0.000, E1  +308.410, E3 -259781.648}
SPL {X  -132.342, Y  +292.599, Z    +0.000, E1  +315.826, E3 -259876.140}
ENDSPLINE

SPLINE
SPL {X  -151.238, Y  +330.309, Z    +0.000, E1  +330.693, E3 -259949.296}
SPL {X  -156.949, Y  +351.453, Z    +0.000, E1  +340.161, E3 -259961.457}
SPL {X  -159.024, Y  +364.945, Z    +0.000, E1  +347.297, E3 -259965.875}
SPL {X  -159.878, Y  +376.512, Z    +0.000, E1  +354.071, E3 -259968.127}
SPL {X  -159.990, Y  +382.403, Z    +0.000, E1  +358.090, E3 -259968.746}
SPL {X  -159.990, Y  +385.261, Z    +0.000, E1  +360.259, E3 -259968.917}
SPL {X  -159.990, Y  +389.002, Z    +0.000, E1  +363.890, E3 -259969.195}
SPL {X  -159.990, Y  +394.493, Z    +0.000, E1  +370.512, E3 -259969.870}
SPL {X  -159.990, Y  +401.377, Z    +0.000, E1  +379.398, E3 -259971.325}
SPL {X  -159.990, Y  +411.365, Z    +0.000, E1  +390.630, E3 -259974.533}
SPL {X  -159.990, Y  +450.467, Z    +0.000, E1  +410.183, E3 -259998.182}
SPL {X  -159.990, Y  +509.934, Z    +0.000, E1  +414.923, E3 -260060.801}
SPL {X  -159.990, Y  +516.848, Z    +0.000, E1  +414.930, E3 -260071.089}
SPL {X  -159.990, Y  +524.818, Z    +0.000, E1  +414.933, E3 -260082.961}
SPL {X  -159.990, Y  +532.100, Z    +0.000, E1  +414.924, E3 -260093.814}
SPL {X  -159.990, Y  +539.391, Z    +0.000, E1  +414.933, E3 -260104.666}
SPL {X  -159.990, Y  +546.283, Z    +0.000, E1  +414.924, E3 -260114.938}
SPL {X  -159.990, Y  +553.734, Z    +0.000, E1  +414.938, E3 -260126.024}
SPL {X  -159.990, Y  +564.956, Z    +0.000, E1  +414.973, E3 -260142.696}
SPL {X  -159.990, Y  +577.902, Z    +0.000, E1  +414.969, E3 -260161.985}
SPL {X  -159.990, Y  +588.063, Z    +0.000, E1  +414.931, E3 -260177.176}
SPL {X  -159.990, Y  +595.273, Z    +0.000, E1  +414.928, E3 -260187.900}
SPL {X  -159.990, Y  +602.326, Z    +0.000, E1  +414.932, E3 -260198.400}
SPL {X  -159.990, Y  +609.708, Z    +0.000, E1  +414.930, E3 -260209.407}
SPL {X  -159.990, Y  +618.088, Z    +0.000, E1  +414.948, E3 -260221.836}
SPL {X  -159.990, Y  +625.928, Z    +0.000, E1  +414.931, E3 -260233.532}
SPL {X  -159.990, Y  +635.803, Z    +0.000, E1  +414.980, E3 -260248.160}
SPL {X  -159.990, Y  +646.303, Z    +0.000, E1  +414.946, E3 -260263.830}
SPL {X  -159.990, Y  +653.312, Z    +0.000, E1  +414.932, E3 -260274.282}
SPL {X  -159.990, Y  +658.943, Z    +0.000, E1  +414.931, E3 -260282.680}
SPL {X  -159.990, Y  +667.151, Z    +0.000, E1  +414.954, E3 -260294.899}
SPL {X  -159.885, Y  +677.285, Z    +0.000, E1  +414.936, E3 -260310.094}
SPL {X  -159.482, Y  +684.244, Z    +0.000, E1  +414.840, E3 -260320.946}
SPL {X  -158.805, Y  +690.934, Z    +0.000, E1  +414.742, E3 -260331.595}
SPL {X  -157.890, Y  +697.337, Z    +0.000, E1  +414.571, E3 -260342.117}
SPL {X  -156.492, Y  +704.774, Z    +0.000, E1  +414.365, E3 -260354.596}
SPL {X  -154.917, Y  +711.470, Z    +0.000, E1  +414.052, E3 -260366.256}
SPL {X  -153.204, Y  +717.603, Z    +0.000, E1  +413.775, E3 -260377.102}
SPL {X  -151.355, Y  +723.351, Z    +0.000, E1  +413.415, E3 -260387.573}
SPL {X  -148.967, Y  +729.859, Z    +0.000, E1  +413.026, E3 -260399.585}
SPL {X  -145.862, Y  +737.236, Z    +0.000, E1  +412.427, E3 -260413.639}
SPL {X  -142.777, Y  +743.691, Z    +0.000, E1  +411.831, E3 -260426.183}
SPL {X  -132.301, Y  +761.463, Z    +0.000, E1  +405.510, E3 -260505.468}
ENDSPLINE

SPLINE
SPL {X  -145.877, Y  +737.201, Z    +0.000, E1  +394.468, E3 -260588.578}
SPL {X  -152.550, Y  +719.721, Z    +0.000, E1  +387.728, E3 -260604.068}
SPL {X  -157.145, Y  +701.536, Z    +0.000, E1  +379.368, E3 -260613.522}
SPL {X  -159.035, Y  +688.952, Z    +0.000, E1  +372.676, E3 -260617.563}
SPL {X  -159.873, Y  +677.622, Z    +0.000, E1  +366.008, E3 -260619.635}
SPL {X  -159.990, Y  +670.381, Z    +0.000, E1  +361.064, E3 -260620.336}
SPL {X  -159.990, Y  +666.603, Z    +0.000, E1  +357.744, E3 -260620.567}
SPL {X  -159.990, Y  +661.750, Z    +0.000, E1  +352.120, E3 -260621.040}
SPL {X  -159.990, Y  +657.656, Z    +0.000, E1  +346.724, E3 -260621.685}
SPL {X  -159.990, Y  +652.023, Z    +0.000, E1  +339.551, E3 -260622.973}
SPL {X  -159.990, Y  +641.935, Z    +0.000, E1  +328.152, E3 -260626.145}
SPL {X  -159.990, Y  +605.095, Z    +0.000, E1  +310.486, E3 -260650.351}
SPL {X  -159.990, Y  +546.155, Z    +0.000, E1  +305.539, E3 -260713.110}
SPL {X  -159.990, Y  +539.348, Z    +0.000, E1  +305.531, E3 -260723.414}
SPL {X  -159.990, Y  +530.752, Z    +0.000, E1  +305.518, E3 -260736.421}
SPL {X  -159.990, Y  +522.797, Z    +0.000, E1  +305.537, E3 -260748.504}
SPL {X  -159.990, Y  +515.332, Z    +0.000, E1  +305.526, E3 -260759.793}
SPL {X  -159.990, Y  +508.047, Z    +0.000, E1  +305.531, E3 -260770.810}
SPL {X  -159.990, Y  +499.403, Z    +0.000, E1  +305.488, E3 -260783.849}
SPL {X  -159.990, Y  +479.413, Z    +0.000, E1  +302.719, E3 -260794.994}
SPL {X  -159.990, Y  +454.926, Z    +0.000, E1  +299.433, E3 -260804.101}
SPL {X  -159.990, Y  +449.697, Z    +0.000, E1  +300.191, E3 -260815.563}
SPL {X  -159.990, Y  +445.847, Z    +0.000, E1  +300.905, E3 -260825.186}
SPL {X  -159.990, Y  +439.266, Z    +0.000, E1  +301.568, E3 -260838.269}
SPL {X  -159.990, Y  +432.883, Z    +0.000, E1  +302.386, E3 -260851.960}
SPL {X  -159.990, Y  +428.299, Z    +0.000, E1  +303.316, E3 -260864.363}
SPL {X  -159.990, Y  +424.402, Z    +0.000, E1  +304.297, E3 -260876.038}
SPL {X  -159.990, Y  +418.562, Z    +0.000, E1  +304.950, E3 -260888.905}
SPL {X  -159.990, Y  +410.722, Z    +0.000, E1  +305.100, E3 -260901.366}
SPL {X  -159.990, Y  +402.790, Z    +0.000, E1  +305.070, E3 -260913.141}
SPL {X  -159.990, Y  +392.953, Z    +0.000, E1  +305.082, E3 -260927.834}
SPL {X  -159.990, Y  +383.354, Z    +0.000, E1  +305.080, E3 -260942.145}
SPL {X  -159.786, Y  +374.425, Z    +0.000, E1  +305.121, E3 -260955.674}
SPL {X  -159.015, Y  +364.863, Z    +0.000, E1  +305.220, E3 -260970.690}
SPL {X  -157.966, Y  +357.131, Z    +0.000, E1  +305.441, E3 -260983.381}
SPL {X  -156.775, Y  +350.586, Z    +0.000, E1  +305.627, E3 -260994.354}
SPL {X  -155.027, Y  +342.959, Z    +0.000, E1  +305.926, E3 -261007.527}
SPL {X  -152.882, Y  +335.340, Z    +0.000, E1  +306.305, E3 -261021.070}
SPL {X  -150.681, Y  +328.723, Z    +0.000, E1  +306.710, E3 -261033.164}
SPL {X  -147.884, Y  +321.449, Z    +0.000, E1  +307.200, E3 -261046.738}
SPL {X  -145.161, Y  +315.232, Z    +0.000, E1  +307.745, E3 -261058.669}
SPL {X  -142.534, Y  +309.830, Z    +0.000, E1  +308.237, E3 -261069.174}
SPL {X  -132.342, Y  +292.599, Z    +0.000, E1  +315.826, E3 -261166.462}
ENDSPLINE

SPLINE
SPL {X  -151.238, Y  +330.309, Z    +0.000, E1  +330.693, E3 -261239.619}
SPL {X  -156.949, Y  +351.453, Z    +0.000, E1  +340.161, E3 -261251.780}
SPL {X  -159.024, Y  +364.945, Z    +0.000, E1  +347.297, E3 -261256.198}
SPL {X  -159.758, Y  +373.891, Z    +0.000, E1  +352.513, E3 -261258.086}
SPL {X  -159.985, Y  +381.208, Z    +0.000, E1  +357.184, E3 -261258.969}
SPL {X  -159.990, Y  +385.261, Z    +0.000, E1  +360.259, E3 -261259.239}
SPL {X  -159.990, Y  +388.094, Z    +0.000, E1  +363.012, E3 -261259.431}
SPL {X  -159.990, Y  +392.053, Z    +0.000, E1  +367.477, E3 -261259.842}
SPL {X  -159.990, Y  +396.158, Z    +0.000, E1  +372.775, E3 -261260.467}
SPL {X  -159.990, Y  +401.377, Z    +0.000, E1  +379.398, E3 -261261.647}
SPL {X  -159.990, Y  +411.365, Z    +0.000, E1  +390.630, E3 -261264.856}
SPL {X  -159.990, Y  +450.467, Z    +0.000, E1  +410.183, E3 -261288.505}
SPL {X  -159.990, Y  +509.934, Z    +0.000, E1  +414.923, E3 -261351.124}
SPL {X  -159.990, Y  +516.848, Z    +0.000, E1  +414.930, E3 -261361.412}
SPL {X  -159.990, Y  +524.818, Z    +0.000, E1  +414.933, E3 -261373.284}
SPL {X  -159.990, Y  +532.100, Z    +0.000, E1  +414.924, E3 -261384.137}
SPL {X  -159.990, Y  +539.391, Z    +0.000, E1  +414.933, E3 -261394.989}
SPL {X  -159.990, Y  +546.283, Z    +0.000, E1  +414.924, E3 -261405.260}
SPL {X  -159.990, Y  +553.734, Z    +0.000, E1  +414.938, E3 -261416.347}
SPL {X  -159.990, Y  +560.657, Z    +0.000, E1  +414.914, E3 -261426.708}
SPL {X  -159.990, Y  +567.311, Z    +0.000, E1  +414.931, E3 -261436.593}
SPL {X  -159.990, Y  +577.902, Z    +0.000, E1  +414.969, E3 -261452.308}
SPL {X  -159.990, Y  +588.063, Z    +0.000, E1  +414.931, E3 -261467.499}
SPL {X  -159.990, Y  +595.273, Z    +0.000, E1  +414.928, E3 -261478.222}
SPL {X  -159.990, Y  +602.326, Z    +0.000, E1  +414.932, E3 -261488.723}
SPL {X  -159.990, Y  +609.708, Z    +0.000, E1  +414.930, E3 -261499.729}
SPL {X  -159.990, Y  +618.088, Z    +0.000, E1  +414.948, E3 -261512.158}
SPL {X  -159.990, Y  +625.928, Z    +0.000, E1  +414.931, E3 -261523.854}
SPL {X  -159.990, Y  +635.803, Z    +0.000, E1  +414.980, E3 -261538.482}
SPL {X  -159.990, Y  +646.303, Z    +0.000, E1  +414.946, E3 -261554.153}
SPL {X  -159.990, Y  +653.312, Z    +0.000, E1  +414.932, E3 -261564.605}
SPL {X  -159.990, Y  +658.943, Z    +0.000, E1  +414.931, E3 -261573.003}
SPL {X  -159.990, Y  +667.151, Z    +0.000, E1  +414.954, E3 -261585.221}
SPL {X  -159.885, Y  +677.285, Z    +0.000, E1  +414.936, E3 -261600.417}
SPL {X  -159.482, Y  +684.244, Z    +0.000, E1  +414.840, E3 -261611.269}
SPL {X  -158.805, Y  +690.934, Z    +0.000, E1  +414.742, E3 -261621.918}
SPL {X  -157.890, Y  +697.337, Z    +0.000, E1  +414.571, E3 -261632.439}
SPL {X  -156.492, Y  +704.774, Z    +0.000, E1  +414.365, E3 -261644.918}
SPL {X  -154.917, Y  +711.470, Z    +0.000, E1  +414.052, E3 -261656.578}
SPL {X  -153.204, Y  +717.603, Z    +0.000, E1  +413.775, E3 -261667.424}
SPL {X  -151.355, Y  +723.351, Z    +0.000, E1  +413.415, E3 -261677.895}
SPL {X  -149.700, Y  +727.952, Z    +0.000, E1  +413.118, E3 -261686.390}
SPL {X  -147.376, Y  +733.767, Z    +0.000, E1  +412.706, E3 -261697.340}
SPL {X  -144.332, Y  +740.529, Z    +0.000, E1  +412.133, E3 -261710.330}
SPL {X  -142.065, Y  +745.081, Z    +0.000, E1  +411.654, E3 -261719.283}
SPL {X  -132.301, Y  +761.463, Z    +0.000, E1  +405.510, E3 -261795.790}
ENDSPLINE

SPLINE
SPL {X  -145.877, Y  +737.201, Z    +0.000, E1  +394.468, E3 -261878.901}
SPL {X  -152.550, Y  +719.721, Z    +0.000, E1  +387.728, E3 -261894.390}
SPL {X  -157.145, Y  +701.536, Z    +0.000, E1  +379.368, E3 -261903.845}
SPL {X  -159.035, Y  +688.952, Z    +0.000, E1  +372.676, E3 -261907.886}
SPL {X  -159.756, Y  +680.154, Z    +0.000, E1  +367.520, E3 -261909.612}
SPL {X  -159.986, Y  +672.560, Z    +0.000, E1  +362.636, E3 -261910.510}
SPL {X  -159.990, Y  +668.344, Z    +0.000, E1  +359.382, E3 -261910.776}
SPL {X  -159.990, Y  +664.070, Z    +0.000, E1  +354.975, E3 -261911.105}
SPL {X  -159.990, Y  +656.953, Z    +0.000, E1  +346.040, E3 -261912.171}
SPL {X  -159.990, Y  +644.589, Z    +0.000, E1  +330.989, E3 -261915.583}
SPL {X  -159.990, Y  +605.095, Z    +0.000, E1  +310.486, E3 -261940.674}
SPL {X  -159.990, Y  +546.155, Z    +0.000, E1  +305.539, E3 -262003.432}
SPL {X  -159.990, Y  +539.348, Z    +0.000, E1  +305.531, E3 -262013.736}
SPL {X  -159.990, Y  +530.752, Z    +0.000, E1  +305.518, E3 -262026.743}
SPL {X  -159.990, Y  +522.797, Z    +0.000, E1  +305.537, E3 -262038.827}
SPL {X  -159.990, Y  +515.332, Z    +0.000, E1  +305.526, E3 -262050.115}
SPL {X  -159.990, Y  +508.047, Z    +0.000, E1  +305.531, E3 -262061.132}
SPL {X  -159.990, Y  +501.296, Z    +0.000, E1  +305.518, E3 -262071.354}
SPL {X  -159.990, Y  +487.558, Z    +0.000, E1  +304.151, E3 -262082.984}
SPL {X  -159.990, Y  +454.926, Z    +0.000, E1  +299.433, E3 -262094.423}
SPL {X  -159.990, Y  +449.697, Z    +0.000, E1  +300.191, E3 -262105.886}
SPL {X  -159.990, Y  +444.026, Z    +0.000, E1  +301.072, E3 -262119.144}
SPL {X  -159.990, Y  +437.596, Z    +0.000, E1  +301.764, E3 -262131.885}
SPL {X  -159.990, Y  +432.883, Z    +0.000, E1  +302.386, E3 -262142.282}
SPL {X  -159.990, Y  +429.044, Z    +0.000, E1  +303.109, E3 -262152.173}
SPL {X  -159.990, Y  +425.222, Z    +0.000, E1  +304.101, E3 -262164.070}
SPL {X  -159.990, Y  +418.562, Z    +0.000, E1  +304.950, E3 -262179.227}
SPL {X  -159.990, Y  +407.911, Z    +0.000, E1  +305.062, E3 -262195.819}
SPL {X  -159.990, Y  +400.284, Z    +0.000, E1  +305.103, E3 -262207.252}
SPL {X  -159.990, Y  +392.953, Z    +0.000, E1  +305.082, E3 -262218.157}
SPL {X  -159.990, Y  +383.354, Z    +0.000, E1  +305.080, E3 -262232.467}
SPL {X  -159.786, Y  +374.425, Z    +0.000, E1  +305.121, E3 -262245.996}
SPL {X  -159.184, Y  +366.462, Z    +0.000, E1  +305.220, E3 -262258.497}
SPL {X  -158.166, Y  +358.413, Z    +0.000, E1  +305.386, E3 -262271.553}
SPL {X  -156.775, Y  +350.586, Z    +0.000, E1  +305.627, E3 -262284.677}
SPL {X  -155.397, Y  +344.442, Z    +0.000, E1  +305.886, E3 -262295.293}
SPL {X  -153.976, Y  +339.046, Z    +0.000, E1  +306.128, E3 -262304.785}
SPL {X  -152.417, Y  +333.859, Z    +0.000, E1  +306.416, E3 -262314.111}
SPL {X  -150.681, Y  +328.723, Z    +0.000, E1  +306.710, E3 -262323.487}
SPL {X  -147.884, Y  +321.449, Z    +0.000, E1  +307.200, E3 -262337.060}
SPL {X  -145.161, Y  +315.232, Z    +0.000, E1  +307.745, E3 -262348.992}
SPL {X  -142.534, Y  +309.830, Z    +0.000, E1  +308.237, E3 -262359.497}
SPL {X  -132.342, Y  +292.599, Z    +0.000, E1  +315.826, E3 -262456.785}
ENDSPLINE

SPLINE
SPL {X  -151.238, Y  +330.309, Z    +0.000, E1  +330.693, E3 -262529.942}
SPL {X  -156.949, Y  +351.453, Z    +0.000, E1  +340.161, E3 -262542.102}
SPL {X  -159.024, Y  +364.945, Z    +0.000, E1  +347.297, E3 -262546.520}
SPL {X  -159.878, Y  +376.512, Z    +0.000, E1  +354.071, E3 -262548.772}
SPL {X  -159.990, Y  +383.659, Z    +0.000, E1  +358.950, E3 -262549.466}
SPL {X  -159.990, Y  +387.327, Z    +0.000, E1  +362.137, E3 -262549.699}
SPL {X  -159.990, Y  +392.053, Z    +0.000, E1  +367.477, E3 -262550.164}
SPL {X  -159.990, Y  +396.158, Z    +0.000, E1  +372.775, E3 -262550.790}
SPL {X  -159.990, Y  +401.377, Z    +0.000, E1  +379.398, E3 -262551.970}
SPL {X  -159.990, Y  +411.365, Z    +0.000, E1  +390.630, E3 -262555.178}
SPL {X  -159.990, Y  +450.467, Z    +0.000, E1  +410.183, E3 -262578.827}
SPL {X  -159.990, Y  +509.934, Z    +0.000, E1  +414.923, E3 -262641.446}
SPL {X  -159.990, Y  +516.848, Z    +0.000, E1  +414.930, E3 -262651.734}
SPL {X  -159.990, Y  +524.818, Z    +0.000, E1  +414.933, E3 -262663.606}
SPL {X  -159.990, Y  +532.100, Z    +0.000, E1  +414.924, E3 -262674.459}
SPL {X  -159.990, Y  +539.391, Z    +0.000, E1  +414.933, E3 -262685.311}
SPL {X  -159.990, Y  +546.283, Z    +0.000, E1  +414.924, E3 -262695.583}
SPL {X  -159.990, Y  +553.734, Z    +0.000, E1  +414.938, E3 -262706.670}
SPL {X  -159.990, Y  +564.956, Z    +0.000, E1  +414.973, E3 -262723.341}
SPL {X  -159.990, Y  +577.902, Z    +0.000, E1  +414.969, E3 -262742.631}
SPL {X  -159.990, Y  +588.063, Z    +0.000, E1  +414.931, E3 -262757.821}
SPL {X  -159.990, Y  +595.273, Z    +0.000, E1  +414.928, E3 -262768.545}
SPL {X  -159.990, Y  +602.326, Z    +0.000, E1  +414.932, E3 -262779.045}
SPL {X  -159.990, Y  +609.708, Z    +0.000, E1  +414.930, E3 -262790.052}
SPL {X  -159.990, Y  +616.306, Z    +0.000, E1  +414.927, E3 -262799.866}
SPL {X  -159.990, Y  +624.320, Z    +0.000, E1  +414.952, E3 -262811.748}
SPL {X  -159.990, Y  +632.991, Z    +0.000, E1  +414.938, E3 -262824.680}
SPL {X  -159.990, Y  +639.033, Z    +0.000, E1  +414.931, E3 -262833.688}
SPL {X  -159.990, Y  +646.303, Z    +0.000, E1  +414.946, E3 -262844.475}
SPL {X  -159.990, Y  +656.335, Z    +0.000, E1  +414.969, E3 -262859.378}
SPL {X  -159.990, Y  +664.577, Z    +0.000, E1  +414.924, E3 -262871.755}
SPL {X  -159.989, Y  +672.128, Z    +0.000, E1  +414.946, E3 -262882.972}
SPL {X  -159.792, Y  +679.466, Z    +0.000, E1  +414.893, E3 -262894.130}
SPL {X  -159.330, Y  +686.016, Z    +0.000, E1  +414.837, E3 -262904.361}
SPL {X  -158.190, Y  +695.432, Z    +0.000, E1  +414.658, E3 -262919.557}
SPL {X  -157.027, Y  +702.151, Z    +0.000, E1  +414.415, E3 -262930.839}
SPL {X  -156.112, Y  +706.513, Z    +0.000, E1  +414.265, E3 -262938.273}
SPL {X  -154.917, Y  +711.470, Z    +0.000, E1  +414.052, E3 -262946.901}
SPL {X  -153.561, Y  +716.398, Z    +0.000, E1  +413.816, E3 -262955.622}
SPL {X  -151.715, Y  +722.287, Z    +0.000, E1  +413.503, E3 -262966.238}
SPL {X  -148.967, Y  +729.859, Z    +0.000, E1  +413.026, E3 -262980.230}
SPL {X  -146.734, Y  +735.264, Z    +0.000, E1  +412.550, E3 -262990.562}
SPL {X  -144.332, Y  +740.529, Z    +0.000, E1  +412.133, E3 -263000.653}
SPL {X  -142.065, Y  +745.081, Z    +0.000, E1  +411.654, E3 -263009.606}
SPL {X  -132.301, Y  +761.463, Z    +0.000, E1  +405.510, E3 -263086.113}
ENDSPLINE

SPLINE
SPL {X  -145.877, Y  +737.201, Z    +0.000, E1  +394.468, E3 -263169.224}
SPL {X  -152.550, Y  +719.721, Z    +0.000, E1  +387.728, E3 -263184.713}
SPL {X  -157.145, Y  +701.536, Z    +0.000, E1  +379.368, E3 -263194.167}
SPL {X  -159.035, Y  +688.952, Z    +0.000, E1  +372.676, E3 -263198.208}
SPL {X  -159.873, Y  +677.622, Z    +0.000, E1  +366.008, E3 -263200.280}
SPL {X  -159.990, Y  +670.381, Z    +0.000, E1  +361.064, E3 -263200.981}
SPL {X  -159.990, Y  +667.647, Z    +0.000, E1  +358.660, E3 -263201.139}
SPL {X  -159.990, Y  +664.070, Z    +0.000, E1  +354.975, E3 -263201.427}
SPL {X  -159.990, Y  +658.737, Z    +0.000, E1  +348.199, E3 -263202.134}
SPL {X  -159.990, Y  +652.023, Z    +0.000, E1  +339.551, E3 -263203.618}
SPL {X  -159.990, Y  +641.935, Z    +0.000, E1  +328.152, E3 -263206.790}
SPL {X  -159.990, Y  +605.095, Z    +0.000, E1  +310.486, E3 -263230.996}
SPL {X  -159.990, Y  +546.155, Z    +0.000, E1  +305.539, E3 -263293.755}
SPL {X  -159.990, Y  +539.348, Z    +0.000, E1  +305.531, E3 -263304.059}
SPL {X  -159.990, Y  +530.752, Z    +0.000, E1  +305.518, E3 -263317.066}
SPL {X  -159.990, Y  +522.797, Z    +0.000, E1  +305.537, E3 -263329.149}
SPL {X  -159.990, Y  +515.332, Z    +0.000, E1  +305.526, E3 -263340.438}
SPL {X  -159.990, Y  +508.047, Z    +0.000, E1  +305.531, E3 -263351.455}
SPL {X  -159.990, Y  +499.403, Z    +0.000, E1  +305.488, E3 -263364.494}
SPL {X  -159.990, Y  +479.413, Z    +0.000, E1  +302.719, E3 -263375.639}
SPL {X  -159.990, Y  +454.926, Z    +0.000, E1  +299.433, E3 -263384.746}
SPL {X  -159.990, Y  +449.697, Z    +0.000, E1  +300.191, E3 -263396.208}
SPL {X  -159.990, Y  +444.026, Z    +0.000, E1  +301.072, E3 -263409.467}
SPL {X  -159.990, Y  +437.596, Z    +0.000, E1  +301.764, E3 -263422.208}
SPL {X  -159.990, Y  +432.883, Z    +0.000, E1  +302.386, E3 -263432.605}
SPL {X  -159.990, Y  +429.044, Z    +0.000, E1  +303.109, E3 -263442.495}
SPL {X  -159.990, Y  +425.222, Z    +0.000, E1  +304.101, E3 -263454.392}
SPL {X  -159.990, Y  +418.562, Z    +0.000, E1  +304.950, E3 -263469.550}
SPL {X  -159.990, Y  +410.722, Z    +0.000, E1  +305.100, E3 -263482.011}
SPL {X  -159.990, Y  +402.790, Z    +0.000, E1  +305.070, E3 -263493.786}
SPL {X  -159.990, Y  +391.119, Z    +0.000, E1  +305.052, E3 -263511.164}
SPL {X  -159.988, Y  +381.720, Z    +0.000, E1  +305.103, E3 -263525.271}
SPL {X  -159.786, Y  +374.425, Z    +0.000, E1  +305.121, E3 -263536.319}
SPL {X  -159.015, Y  +364.863, Z    +0.000, E1  +305.220, E3 -263551.335}
SPL {X  -157.966, Y  +357.131, Z    +0.000, E1  +305.441, E3 -263564.026}
SPL {X  -156.775, Y  +350.586, Z    +0.000, E1  +305.627, E3 -263575.000}
SPL {X  -155.397, Y  +344.442, Z    +0.000, E1  +305.886, E3 -263585.615}
SPL {X  -153.976, Y  +339.046, Z    +0.000, E1  +306.128, E3 -263595.108}
SPL {X  -152.417, Y  +333.859, Z    +0.000, E1  +306.416, E3 -263604.434}
SPL {X  -150.681, Y  +328.723, Z    +0.000, E1  +306.710, E3 -263613.810}
SPL {X  -147.884, Y  +321.449, Z    +0.000, E1  +307.200, E3 -263627.383}
SPL {X  -145.161, Y  +315.232, Z    +0.000, E1  +307.745, E3 -263639.314}
SPL {X  -142.534, Y  +309.830, Z    +0.000, E1  +308.237, E3 -263649.819}
SPL {X  -132.342, Y  +292.599, Z    +0.000, E1  +315.826, E3 -263747.107}
ENDSPLINE

SPLINE
SPL {X  -151.238, Y  +330.309, Z    +0.000, E1  +330.693, E3 -263820.264}
SPL {X  -156.949, Y  +351.453, Z    +0.000, E1  +340.161, E3 -263832.425}
SPL {X  -159.024, Y  +364.945, Z    +0.000, E1  +347.297, E3 -263836.843}
SPL {X  -159.758, Y  +373.891, Z    +0.000, E1  +352.513, E3 -263838.732}
SPL {X  -159.985, Y  +381.208, Z    +0.000, E1  +357.184, E3 -263839.614}
SPL {X  -159.990, Y  +384.493, Z    +0.000, E1  +359.676, E3 -263839.839}
SPL {X  -159.990, Y  +387.327, Z    +0.000, E1  +362.137, E3 -263840.022}
SPL {X  -159.990, Y  +392.053, Z    +0.000, E1  +367.477, E3 -263840.487}
SPL {X  -159.990, Y  +396.158, Z    +0.000, E1  +372.775, E3 -263841.112}
SPL {X  -159.990, Y  +401.377, Z    +0.000, E1  +379.398, E3 -263842.293}
SPL {X  -159.990, Y  +411.365, Z    +0.000, E1  +390.630, E3 -263845.501}
SPL {X  -159.990, Y  +450.467, Z    +0.000, E1  +410.183, E3 -263869.150}
SPL {X  -159.990, Y  +509.934, Z    +0.000, E1  +414.923, E3 -263931.769}
SPL {X  -159.990, Y  +516.848, Z    +0.000, E1  +414.930, E3 -263942.057}
SPL {X  -159.990, Y  +524.818, Z    +0.000, E1  +414.933, E3 -263953.929}
SPL {X  -159.990, Y  +532.100, Z    +0.000, E1  +414.924, E3 -263964.782}
SPL {X  -159.990, Y  +539.391, Z    +0.000, E1  +414.933, E3 -263975.634}
SPL {X  -159.990, Y  +546.283, Z    +0.000, E1  +414.924, E3 -263985.905}
SPL {X  -159.990, Y  +553.734, Z    +0.000, E1  +414.938, E3 -263996.992}
SPL {X  -159.990, Y  +564.956, Z    +0.000, E1  +414.973, E3 -264013.663}
SPL {X  -159.990, Y  +577.902, Z    +0.000, E1  +414.969, E3 -264032.953}
SPL {X  -159.990, Y  +588.063, Z    +0.000, E1  +414.931, E3 -264048.144}
SPL {X  -159.990, Y  +595.273, Z    +0.000, E1  +414.928, E3 -264058.868}
SPL {X  -159.990, Y  +602.326, Z    +0.000, E1  +414.932, E3 -264069.368}
SPL {X  -159.990, Y  +609.708, Z    +0.000, E1  +414.930, E3 -264080.375}
SPL {X  -159.990, Y  +618.088, Z    +0.000, E1  +414.948, E3 -264092.804}
SPL {X  -159.990, Y  +625.928, Z    +0.000, E1  +414.931, E3 -264104.499}
SPL {X  -159.990, Y  +635.803, Z    +0.000, E1  +414.980, E3 -264119.128}
SPL {X  -159.990, Y  +646.303, Z    +0.000, E1  +414.946, E3 -264134.798}
SPL {X  -159.990, Y  +653.312, Z    +0.000, E1  +414.932, E3 -264145.250}
SPL {X  -159.990, Y  +661.828, Z    +0.000, E1  +414.965, E3 -264157.906}
SPL {X  -159.989, Y  +672.128, Z    +0.000, E1  +414.946, E3 -264173.294}
SPL {X  -159.636, Y  +682.136, Z    +0.000, E1  +414.901, E3 -264188.552}
SPL {X  -158.805, Y  +690.934, Z    +0.000, E1  +414.742, E3 -264202.563}
SPL {X  -157.512, Y  +699.550, Z    +0.000, E1  +414.543, E3 -264216.714}
SPL {X  -156.112, Y  +706.513, Z    +0.000, E1  +414.265, E3 -264228.596}
SPL {X  -154.917, Y  +711.470, Z    +0.000, E1  +414.052, E3 -264237.223}
SPL {X  -153.561, Y  +716.398, Z    +0.000, E1  +413.816, E3 -264245.945}
SPL {X  -151.715, Y  +722.287, Z    +0.000, E1  +413.503, E3 -264256.561}
SPL {X  -149.700, Y  +727.952, Z    +0.000, E1  +413.118, E3 -264267.035}
SPL {X  -147.376, Y  +733.767, Z    +0.000, E1  +412.706, E3 -264277.985}
SPL {X  -145.109, Y  +738.881, Z    +0.000, E1  +412.243, E3 -264287.832}
SPL {X  -142.777, Y  +743.691, Z    +0.000, E1  +411.831, E3 -264297.150}
SPL {X  -132.301, Y  +761.463, Z    +0.000, E1  +405.510, E3 -264376.435}
ENDSPLINE

SPLINE
SPL {X  -145.877, Y  +737.201, Z    +0.000, E1  +394.468, E3 -264459.546}
SPL {X  -152.550, Y  +719.721, Z    +0.000, E1  +387.728, E3 -264475.035}
SPL {X  -157.145, Y  +701.536, Z    +0.000, E1  +379.368, E3 -264484.490}
SPL {X  -159.035, Y  +688.952, Z    +0.000, E1  +372.676, E3 -264488.531}
SPL {X  -159.756, Y  +680.154, Z    +0.000, E1  +367.520, E3 -264490.257}
SPL {X  -159.986, Y  +672.560, Z    +0.000, E1  +362.636, E3 -264491.155}
SPL {X  -159.990, Y  +668.344, Z    +0.000, E1  +359.382, E3 -264491.422}
SPL {X  -159.990, Y  +664.070, Z    +0.000, E1  +354.975, E3 -264491.750}
SPL {X  -159.990, Y  +656.953, Z    +0.000, E1  +346.040, E3 -264492.817}
SPL {X  -159.990, Y  +644.589, Z    +0.000, E1  +330.989, E3 -264496.228}
SPL {X  -159.990, Y  +605.095, Z    +0.000, E1  +310.486, E3 -264521.319}
SPL {X  -159.990, Y  +546.155, Z    +0.000, E1  +305.539, E3 -264584.077}
SPL {X  -159.990, Y  +539.348, Z    +0.000, E1  +305.531, E3 -264594.381}
SPL {X  -159.990, Y  +530.752, Z    +0.000, E1  +305.518, E3 -264607.389}
SPL {X  -159.990, Y  +522.797, Z    +0.000, E1  +305.537, E3 -264619.472}
SPL {X  -159.990, Y  +515.332, Z    +0.000, E1  +305.526, E3 -264630.761}
SPL {X  -159.990, Y  +508.047, Z    +0.000, E1  +305.531, E3 -264641.777}
SPL {X  -159.990, Y  +501.296, Z    +0.000, E1  +305.518, E3 -264651.999}
SPL {X  -159.990, Y  +487.558, Z    +0.000, E1  +304.151, E3 -264663.629}
SPL {X  -159.990, Y  +454.926, Z    +0.000, E1  +299.433, E3 -264675.068}
SPL {X  -159.990, Y  +449.697, Z    +0.000, E1  +300.191, E3 -264686.531}
SPL {X  -159.990, Y  +445.847, Z    +0.000, E1  +300.905, E3 -264696.154}
SPL {X  -159.990, Y  +439.266, Z    +0.000, E1  +301.568, E3 -264709.237}
SPL {X  -159.990, Y  +432.883, Z    +0.000, E1  +302.386, E3 -264722.927}
SPL {X  -159.990, Y  +429.044, Z    +0.000, E1  +303.109, E3 -264732.818}
SPL {X  -159.990, Y  +425.222, Z    +0.000, E1  +304.101, E3 -264744.715}
SPL {X  -159.990, Y  +420.083, Z    +0.000, E1  +304.918, E3 -264757.291}
SPL {X  -159.990, Y  +412.567, Z    +0.000, E1  +305.072, E3 -264769.515}
SPL {X  -159.990, Y  +405.235, Z    +0.000, E1  +305.098, E3 -264780.503}
SPL {X  -159.990, Y  +400.284, Z    +0.000, E1  +305.103, E3 -264787.898}
SPL {X  -159.990, Y  +391.119, Z    +0.000, E1  +305.052, E3 -264801.486}
SPL {X  -159.988, Y  +381.720, Z    +0.000, E1  +305.103, E3 -264815.593}
SPL {X  -159.786, Y  +374.425, Z    +0.000, E1  +305.121, E3 -264826.642}
SPL {X  -159.184, Y  +366.462, Z    +0.000, E1  +305.220, E3 -264839.142}
SPL {X  -158.166, Y  +358.413, Z    +0.000, E1  +305.386, E3 -264852.198}
SPL {X  -156.775, Y  +350.586, Z    +0.000, E1  +305.627, E3 -264865.322}
SPL {X  -155.027, Y  +342.959, Z    +0.000, E1  +305.926, E3 -264878.495}
SPL {X  -152.882, Y  +335.340, Z    +0.000, E1  +306.305, E3 -264892.038}
SPL {X  -150.681, Y  +328.723, Z    +0.000, E1  +306.710, E3 -264904.132}
SPL {X  -147.884, Y  +321.449, Z    +0.000, E1  +307.200, E3 -264917.705}
SPL {X  -144.518, Y  +313.862, Z    +0.000, E1  +307.832, E3 -264932.251}
SPL {X  -141.812, Y  +308.430, Z    +0.000, E1  +308.410, E3 -264942.938}
SPL {X  -132.342, Y  +292.599, Z    +0.000, E1  +315.826, E3 -265037.430}
ENDSPLINE

SPLINE
SPL {X  -151.238, Y  +330.309, Z    +0.000, E1  +330.693, E3 -265110.587}
SPL {X  -156.949, Y  +351.453, Z    +0.000, E1  +340.161, E3 -265122.748}
SPL {X  -159.024, Y  +364.945, Z    +0.000, E1  +347.297, E3 -265127.165}
SPL {X  -159.758, Y  +373.891, Z    +0.000, E1  +352.513, E3 -265129.054}
SPL {X  -159.985, Y  +381.208, Z    +0.000, E1  +357.184, E3 -265129.937}
SPL {X  -159.990, Y  +384.493, Z    +0.000, E1  +359.676, E3 -265130.162}
SPL {X  -159.990, Y  +387.327, Z    +0.000, E1  +362.137, E3 -265130.344}
SPL {X  -159.990, Y  +392.053, Z    +0.000, E1  +367.477, E3 -265130.809}
SPL {X  -159.990, Y  +396.158, Z    +0.000, E1  +372.775, E3 -265131.435}
SPL {X  -159.990, Y  +401.377, Z    +0.000, E1  +379.398, E3 -265132.615}
SPL {X  -159.990, Y  +411.365, Z    +0.000, E1  +390.630, E3 -265135.824}
SPL {X  -159.990, Y  +450.467, Z    +0.000, E1  +410.183, E3 -265159.472}
SPL {X  -159.990, Y  +509.934, Z    +0.000, E1  +414.923, E3 -265222.091}
SPL {X  -159.990, Y  +516.848, Z    +0.000, E1  +414.930, E3 -265232.379}
SPL {X  -159.990, Y  +524.818, Z    +0.000, E1  +414.933, E3 -265244.251}
SPL {X  -159.990, Y  +532.100, Z    +0.000, E1  +414.924, E3 -265255.104}
SPL {X  -159.990, Y  +539.391, Z    +0.000, E1  +414.933, E3 -265265.956}
SPL {X  -159.990, Y  +546.283, Z    +0.000, E1  +414.924, E3 -265276.228}
SPL {X  -159.990, Y  +553.734, Z    +0.000, E1  +414.938, E3 -265287.315}
SPL {X  -159.990, Y  +564.956, Z    +0.000, E1  +414.973, E3 -265303.986}
SPL {X  -159.990, Y  +577.902, Z    +0.000, E1  +414.969, E3 -265323.276}
SPL {X  -159.990, Y  +588.063, Z    +0.000, E1  +414.931, E3 -265338.467}
SPL {X  -159.990, Y  +595.273, Z    +0.000, E1  +414.928, E3 -265349.190}
SPL {X  -159.990, Y  +602.326, Z    +0.000, E1  +414.932, E3 -265359.691}
SPL {X  -159.990, Y  +609.708, Z    +0.000, E1  +414.930, E3 -265370.697}
SPL {X  -159.990, Y  +618.088, Z    +0.000, E1  +414.948, E3 -265383.126}
SPL {X  -159.990, Y  +625.928, Z    +0.000, E1  +414.931, E3 -265394.822}
SPL {X  -159.990, Y  +635.803, Z    +0.000, E1  +414.980, E3 -265409.450}
SPL {X  -159.990, Y  +646.303, Z    +0.000, E1  +414.946, E3 -265425.121}
SPL {X  -159.990, Y  +656.335, Z    +0.000, E1  +414.969, E3 -265440.023}
SPL {X  -159.990, Y  +664.577, Z    +0.000, E1  +414.924, E3 -265452.400}
SPL {X  -159.989, Y  +672.128, Z    +0.000, E1  +414.946, E3 -265463.617}
SPL {X  -159.636, Y  +682.136, Z    +0.000, E1  +414.901, E3 -265478.875}
SPL {X  -158.805, Y  +690.934, Z    +0.000, E1  +414.742, E3 -265492.886}
SPL {X  -157.890, Y  +697.337, Z    +0.000, E1  +414.571, E3 -265503.407}
SPL {X  -156.492, Y  +704.774, Z    +0.000, E1  +414.365, E3 -265515.886}
SPL {X  -154.917, Y  +711.470, Z    +0.000, E1  +414.052, E3 -265527.546}
SPL {X  -153.204, Y  +717.603, Z    +0.000, E1  +413.775, E3 -265538.392}
SPL {X  -151.355, Y  +723.351, Z    +0.000, E1  +413.415, E3 -265548.863}
SPL {X  -148.967, Y  +729.859, Z    +0.000, E1  +413.026, E3 -265560.875}
SPL {X  -145.862, Y  +737.236, Z    +0.000, E1  +412.427, E3 -265574.930}
SPL {X  -142.777, Y  +743.691, Z    +0.000, E1  +411.831, E3 -265587.473}
SPL {X  -132.301, Y  +761.463, Z    +0.000, E1  +405.510, E3 -265666.758}
ENDSPLINE

SPLINE
SPL {X  -145.877, Y  +737.201, Z    +0.000, E1  +394.468, E3 -265749.869}
SPL {X  -152.550, Y  +719.721, Z    +0.000, E1  +387.728, E3 -265765.358}
SPL {X  -157.145, Y  +701.536, Z    +0.000, E1  +379.368, E3 -265774.813}
SPL {X  -159.035, Y  +688.952, Z    +0.000, E1  +372.676, E3 -265778.854}
SPL {X  -159.756, Y  +680.154, Z    +0.000, E1  +367.520, E3 -265780.580}
SPL {X  -159.986, Y  +672.560, Z    +0.000, E1  +362.636, E3 -265781.478}
SPL {X  -159.990, Y  +669.364, Z    +0.000, E1  +360.170, E3 -265781.686}
SPL {X  -159.990, Y  +667.647, Z    +0.000, E1  +358.660, E3 -265781.784}
SPL {X  -159.990, Y  +664.070, Z    +0.000, E1  +354.975, E3 -265782.073}
SPL {X  -159.990, Y  +656.953, Z    +0.000, E1  +346.040, E3 -265783.139}
SPL {X  -159.990, Y  +644.589, Z    +0.000, E1  +330.989, E3 -265786.551}
SPL {X  -159.990, Y  +605.095, Z    +0.000, E1  +310.486, E3 -265811.641}
SPL {X  -159.990, Y  +546.155, Z    +0.000, E1  +305.539, E3 -265874.400}
SPL {X  -159.990, Y  +539.348, Z    +0.000, E1  +305.531, E3 -265884.704}
SPL {X  -159.990, Y  +530.752, Z    +0.000, E1  +305.518, E3 -265897.711}
SPL {X  -159.990, Y  +522.797, Z    +0.000, E1  +305.537, E3 -265909.794}
SPL {X  -159.990, Y  +515.332, Z    +0.000, E1  +305.526, E3 -265921.083}
SPL {X  -159.990, Y  +508.047, Z    +0.000, E1  +305.531, E3 -265932.100}
SPL {X  -159.990, Y  +499.403, Z    +0.000, E1  +305.488, E3 -265945.139}
SPL {X  -159.990, Y  +479.413, Z    +0.000, E1  +302.719, E3 -265956.284}
SPL {X  -159.990, Y  +454.926, Z    +0.000, E1  +299.433, E3 -265965.391}
SPL {X  -159.990, Y  +449.697, Z    +0.000, E1  +300.191, E3 -265976.853}
SPL {X  -159.990, Y  +445.847, Z    +0.000, E1  +300.905, E3 -265986.476}
SPL {X  -159.990, Y  +439.266, Z    +0.000, E1  +301.568, E3 -265999.560}
SPL {X  -159.990, Y  +432.883, Z    +0.000, E1  +302.386, E3 -266013.250}
SPL {X  -159.990, Y  +429.044, Z    +0.000, E1  +303.109, E3 -266023.140}
SPL {X  -159.990, Y  +425.222, Z    +0.000, E1  +304.101, E3 -266035.037}
SPL {X  -159.990, Y  +420.083, Z    +0.000, E1  +304.918, E3 -266047.613}
SPL {X  -159.990, Y  +412.567, Z    +0.000, E1  +305.072, E3 -266059.837}
SPL {X  -159.990, Y  +402.790, Z    +0.000, E1  +305.070, E3 -266074.431}
SPL {X  -159.990, Y  +391.119, Z    +0.000, E1  +305.052, E3 -266091.809}
SPL {X  -159.988, Y  +381.720, Z    +0.000, E1  +305.103, E3 -266105.916}
SPL {X  -159.786, Y  +374.425, Z    +0.000, E1  +305.121, E3 -266116.964}
SPL {X  -159.015, Y  +364.863, Z    +0.000, E1  +305.220, E3 -266131.980}
SPL {X  -157.966, Y  +357.131, Z    +0.000, E1  +305.441, E3 -266144.671}
SPL {X  -156.775, Y  +350.586, Z    +0.000, E1  +305.627, E3 -266155.645}
SPL {X  -155.027, Y  +342.959, Z    +0.000, E1  +305.926, E3 -266168.818}
SPL {X  -152.882, Y  +335.340, Z    +0.000, E1  +306.305, E3 -266182.360}
SPL {X  -150.681, Y  +328.723, Z    +0.000, E1  +306.710, E3 -266194.455}
SPL {X  -148.661, Y  +323.366, Z    +0.000, E1  +307.100, E3 -266204.464}
SPL {X  -147.089, Y  +319.560, Z    +0.000, E1  +307.396, E3 -266211.679}
SPL {X  -145.161, Y  +315.232, Z    +0.000, E1  +307.745, E3 -266219.959}
SPL {X  -142.534, Y  +309.830, Z    +0.000, E1  +308.237, E3 -266230.465}
SPL {X  -132.342, Y  +292.599, Z    +0.000, E1  +315.826, E3 -266327.753}
ENDSPLINE

SPLINE
SPL {X  -151.238, Y  +330.309, Z    +0.000, E1  +330.693, E3 -266400.909}
SPL {X  -156.949, Y  +351.453, Z    +0.000, E1  +340.161, E3 -266413.070}
SPL {X  -159.024, Y  +364.945, Z    +0.000, E1  +347.297, E3 -266417.488}
SPL {X  -159.878, Y  +376.512, Z    +0.000, E1  +354.071, E3 -266419.739}
SPL {X  -159.990, Y  +383.659, Z    +0.000, E1  +358.950, E3 -266420.434}
SPL {X  -159.990, Y  +387.327, Z    +0.000, E1  +362.137, E3 -266420.667}
SPL {X  -159.990, Y  +390.622, Z    +0.000, E1  +365.876, E3 -266420.960}
SPL {X  -159.990, Y  +394.493, Z    +0.000, E1  +370.512, E3 -266421.483}
SPL {X  -159.990, Y  +401.377, Z    +0.000, E1  +379.398, E3 -266422.938}
SPL {X  -159.990, Y  +411.365, Z    +0.000, E1  +390.630, E3 -266426.146}
SPL {X  -159.990, Y  +450.467, Z    +0.000, E1  +410.183, E3 -266449.795}
SPL {X  -159.990, Y  +509.934, Z    +0.000, E1  +414.923, E3 -266512.414}
SPL {X  -159.990, Y  +516.848, Z    +0.000, E1  +414.930, E3 -266522.702}
SPL {X  -159.990, Y  +524.818, Z    +0.000, E1  +414.933, E3 -266534.574}
SPL {X  -159.990, Y  +532.100, Z    +0.000, E1  +414.924, E3 -266545.427}
SPL {X  -159.990, Y  +539.391, Z    +0.000, E1  +414.933, E3 -266556.279}
SPL {X  -159.990, Y  +546.283, Z    +0.000, E1  +414.924, E3 -266566.551}
SPL {X  -159.990, Y  +553.734, Z    +0.000, E1  +414.938, E3 -266577.637}
SPL {X  -159.990, Y  +564.956, Z    +0.000, E1  +414.973, E3 -266594.309}
SPL {X  -159.990, Y  +577.902, Z    +0.000, E1  +414.969, E3 -266613.598}
SPL {X  -159.990, Y  +588.063, Z    +0.000, E1  +414.931, E3 -266628.789}
SPL {X  -159.990, Y  +595.273, Z    +0.000, E1  +414.928, E3 -266639.513}
SPL {X  -159.990, Y  +602.326, Z    +0.000, E1  +414.932, E3 -266650.013}
SPL {X  -159.990, Y  +609.708, Z    +0.000, E1  +414.930, E3 -266661.020}
SPL {X  -159.990, Y  +618.088, Z    +0.000, E1  +414.948, E3 -266673.449}
SPL {X  -159.990, Y  +625.928, Z    +0.000, E1  +414.931, E3 -266685.145}
SPL {X  -159.990, Y  +635.803, Z    +0.000, E1  +414.980, E3 -266699.773}
SPL {X  -159.990, Y  +646.303, Z    +0.000, E1  +414.946, E3 -266715.443}
SPL {X  -159.990, Y  +653.312, Z    +0.000, E1  +414.932, E3 -266725.895}
SPL {X  -159.990, Y  +658.943, Z    +0.000, E1  +414.931, E3 -266734.293}
SPL {X  -159.990, Y  +667.151, Z    +0.000, E1  +414.954, E3 -266746.512}
SPL {X  -159.885, Y  +677.285, Z    +0.000, E1  +414.936, E3 -266761.707}
SPL {X  -159.482, Y  +684.244, Z    +0.000, E1  +414.840, E3 -266772.559}
SPL {X  -158.805, Y  +690.934, Z    +0.000, E1  +414.742, E3 -266783.208}
SPL {X  -157.890, Y  +697.337, Z    +0.000, E1  +414.571, E3 -266793.730}
SPL {X  -156.492, Y  +704.774, Z    +0.000, E1  +414.365, E3 -266806.209}
SPL {X  -154.917, Y  +711.470, Z    +0.000, E1  +414.052, E3 -266817.868}
SPL {X  -153.561, Y  +716.398, Z    +0.000, E1  +413.816, E3 -266826.590}
SPL {X  -151.715, Y  +722.287, Z    +0.000, E1  +413.503, E3 -266837.206}
SPL {X  -148.967, Y  +729.859, Z    +0.000, E1  +413.026, E3 -266851.198}
SPL {X  -145.862, Y  +737.236, Z    +0.000, E1  +412.427, E3 -266865.252}
SPL {X  -142.777, Y  +743.691, Z    +0.000, E1  +411.831, E3 -266877.795}
SPL {X  -132.301, Y  +761.463, Z    +0.000, E1  +405.510, E3 -266957.080}
ENDSPLINE

